KUKA KRL program: unicorn2_2.src

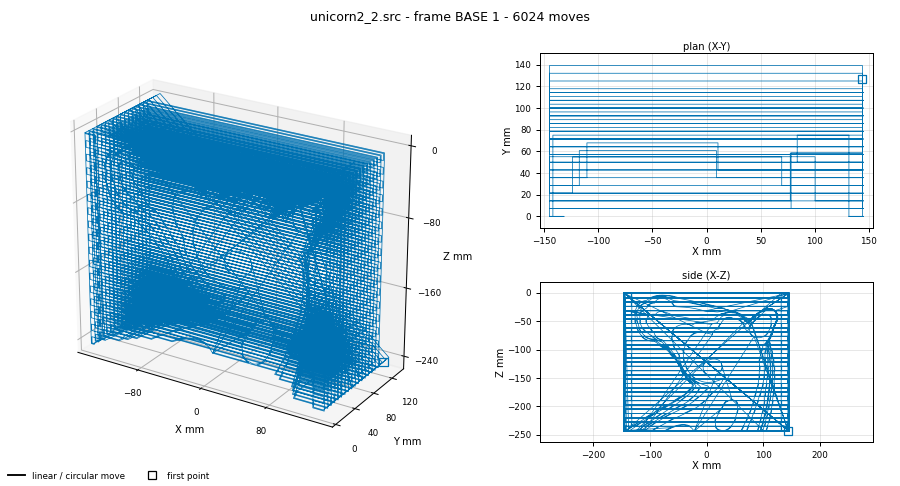
[picture p0: tool path of unicorn2_2.src in frame BASE 1, 6024 of 6025 moves have a stored position in this frame; points joined in program order, loops and branches not executed]
&ACCESS RVP
&REL 1
&PARAM TEMPLATE = C:\KRC\Roboter\Template\vorgabe
&PARAM EDITMASK = *
DEF unicorn2_2( )
EXT BAS (BAS_COMMAND :IN,REAL :IN )

INT INDX
FOR INDX=1 TO 6
	$ACC_AXIS[INDX]=50
	$VEL_AXIS[INDX]=20
ENDFOR

$VEL.ORI1=200
$VEL.ORI2=200
$ACC.ORI1=100
$ACC.ORI2=100

$VEL.CP = 0.2
$ACC.CP = 5

$IPO_MODE = #BASE
$APO.CDIS = 0.5
$ADVANCE = 5

$ACT_TOOL = 1
$TOOL=TOOL_DATA[1]
$ACT_BASE = 1
$BASE=BASE_DATA[1]

PTP {A1 -30.0,A2 -90.0,A3 90.0,A4 0.0,A5 90.0,A6 0.0}

LIN {X 144.015,Y 126.800,Z -242.561,A 90.000,B 90.000,C 0.000} C_DIS
LIN {X 144.015,Y 114.300,Z -242.561,A 90.000,B 90.000,C 0.000} C_DIS
LIN {X -144.015,Y 114.300,Z -242.561,A 90.000,B 90.000,C 0.000} C_DIS
LIN {X -144.015,Y 114.300,Z -235.012,A 90.000,B 90.000,C 0.000} C_DIS
LIN {X 144.015,Y 114.300,Z -235.012,A 90.000,B 90.000,C 0.000} C_DIS
LIN {X 144.015,Y 114.300,Z -227.464,A 90.000,B 90.000,C 0.000} C_DIS
LIN {X -144.015,Y 114.300,Z -227.464,A 90.000,B 90.000,C 0.000} C_DIS
LIN {X -144.015,Y 114.300,Z -219.915,A 90.000,B 90.000,C 0.000} C_DIS
LIN {X 144.015,Y 114.300,Z -219.915,A 90.000,B 90.000,C 0.000} C_DIS
LIN {X 144.015,Y 114.300,Z -212.366,A 90.000,B 90.000,C 0.000} C_DIS
LIN {X -144.015,Y 114.300,Z -212.366,A 90.000,B 90.000,C 0.000} C_DIS
LIN {X -144.015,Y 114.300,Z -204.817,A 90.000,B 90.000,C 0.000} C_DIS
LIN {X 144.015,Y 114.300,Z -204.817,A 90.000,B 90.000,C 0.000} C_DIS
LIN {X 144.015,Y 114.300,Z -197.269,A 90.000,B 90.000,C 0.000} C_DIS
LIN {X -144.015,Y 114.300,Z -197.269,A 90.000,B 90.000,C 0.000} C_DIS
LIN {X -144.015,Y 114.300,Z -189.720,A 90.000,B 90.000,C 0.000} C_DIS
LIN {X 144.015,Y 114.300,Z -189.720,A 90.000,B 90.000,C 0.000} C_DIS
LIN {X 144.015,Y 114.300,Z -182.171,A 90.000,B 90.000,C 0.000} C_DIS
LIN {X -144.015,Y 114.300,Z -182.171,A 90.000,B 90.000,C 0.000} C_DIS
LIN {X -144.015,Y 114.300,Z -174.622,A 90.000,B 90.000,C 0.000} C_DIS
LIN {X 144.015,Y 114.300,Z -174.622,A 90.000,B 90.000,C 0.000} C_DIS
LIN {X 144.015,Y 114.300,Z -167.073,A 90.000,B 90.000,C 0.000} C_DIS
LIN {X -144.015,Y 114.300,Z -167.073,A 90.000,B 90.000,C 0.000} C_DIS
LIN {X -144.015,Y 114.300,Z -159.525,A 90.000,B 90.000,C 0.000} C_DIS
LIN {X 144.015,Y 114.300,Z -159.525,A 90.000,B 90.000,C 0.000} C_DIS
LIN {X 144.015,Y 114.300,Z -151.976,A 90.000,B 90.000,C 0.000} C_DIS
LIN {X -144.015,Y 114.300,Z -151.976,A 90.000,B 90.000,C 0.000} C_DIS
LIN {X -144.015,Y 114.300,Z -144.427,A 90.000,B 90.000,C 0.000} C_DIS
LIN {X 144.015,Y 114.300,Z -144.427,A 90.000,B 90.000,C 0.000} C_DIS
LIN {X 144.015,Y 114.300,Z -136.878,A 90.000,B 90.000,C 0.000} C_DIS
LIN {X -144.015,Y 114.300,Z -136.878,A 90.000,B 90.000,C 0.000} C_DIS
LIN {X -144.015,Y 114.300,Z -129.329,A 90.000,B 90.000,C 0.000} C_DIS
LIN {X 144.015,Y 114.300,Z -129.329,A 90.000,B 90.000,C 0.000} C_DIS
LIN {X 144.015,Y 114.300,Z -121.781,A 90.000,B 90.000,C 0.000} C_DIS
LIN {X -144.015,Y 114.300,Z -121.781,A 90.000,B 90.000,C 0.000} C_DIS
LIN {X -144.015,Y 114.300,Z -114.232,A 90.000,B 90.000,C 0.000} C_DIS
LIN {X 144.015,Y 114.300,Z -114.232,A 90.000,B 90.000,C 0.000} C_DIS
LIN {X 144.015,Y 114.300,Z -106.683,A 90.000,B 90.000,C 0.000} C_DIS
LIN {X -144.015,Y 114.300,Z -106.683,A 90.000,B 90.000,C 0.000} C_DIS
LIN {X -144.015,Y 114.300,Z -99.134,A 90.000,B 90.000,C 0.000} C_DIS
LIN {X 144.015,Y 114.300,Z -99.134,A 90.000,B 90.000,C 0.000} C_DIS
LIN {X 144.015,Y 114.300,Z -91.586,A 90.000,B 90.000,C 0.000} C_DIS
LIN {X -144.015,Y 114.300,Z -91.586,A 90.000,B 90.000,C 0.000} C_DIS
LIN {X -144.015,Y 114.300,Z -84.037,A 90.000,B 90.000,C 0.000} C_DIS
LIN {X 144.015,Y 114.300,Z -84.037,A 90.000,B 90.000,C 0.000} C_DIS
LIN {X 144.015,Y 114.300,Z -76.488,A 90.000,B 90.000,C 0.000} C_DIS
LIN {X -144.015,Y 114.300,Z -76.488,A 90.000,B 90.000,C 0.000} C_DIS
LIN {X -144.015,Y 114.300,Z -68.939,A 90.000,B 90.000,C 0.000} C_DIS
LIN {X 144.015,Y 114.300,Z -68.939,A 90.000,B 90.000,C 0.000} C_DIS
LIN {X 144.015,Y 114.300,Z -61.390,A 90.000,B 90.000,C 0.000} C_DIS
LIN {X -144.015,Y 114.300,Z -61.390,A 90.000,B 90.000,C 0.000} C_DIS
LIN {X -144.015,Y 114.300,Z -53.842,A 90.000,B 90.000,C 0.000} C_DIS
LIN {X 144.015,Y 114.300,Z -53.842,A 90.000,B 90.000,C 0.000} C_DIS
LIN {X 144.015,Y 114.300,Z -46.293,A 90.000,B 90.000,C 0.000} C_DIS
LIN {X -144.015,Y 114.300,Z -46.293,A 90.000,B 90.000,C 0.000} C_DIS
LIN {X -144.015,Y 114.300,Z -38.744,A 90.000,B 90.000,C 0.000} C_DIS
LIN {X 144.015,Y 114.300,Z -38.744,A 90.000,B 90.000,C 0.000} C_DIS
LIN {X 144.015,Y 114.300,Z -31.195,A 90.000,B 90.000,C 0.000} C_DIS
LIN {X -144.015,Y 114.300,Z -31.195,A 90.000,B 90.000,C 0.000} C_DIS
LIN {X -144.015,Y 114.300,Z -23.646,A 90.000,B 90.000,C 0.000} C_DIS
LIN {X 144.015,Y 114.300,Z -23.646,A 90.000,B 90.000,C 0.000} C_DIS
LIN {X 144.015,Y 114.300,Z -16.098,A 90.000,B 90.000,C 0.000} C_DIS
LIN {X -144.015,Y 114.300,Z -16.098,A 90.000,B 90.000,C 0.000} C_DIS
LIN {X -144.015,Y 114.300,Z -8.549,A 90.000,B 90.000,C 0.000} C_DIS
LIN {X 144.015,Y 114.300,Z -8.549,A 90.000,B 90.000,C 0.000} C_DIS
LIN {X 144.015,Y 114.300,Z -1.000,A 90.000,B 90.000,C 0.000} C_DIS
LIN {X -144.015,Y 114.300,Z -1.000,A 90.000,B 90.000,C 0.000} C_DIS
LIN {X -145.015,Y 114.300,Z 0.000,A 90.000,B 90.000,C 0.000} C_DIS
LIN {X 145.015,Y 114.300,Z 0.000,A 90.000,B 90.000,C 0.000} C_DIS
LIN {X 145.015,Y 114.300,Z -243.561,A 90.000,B 90.000,C 0.000} C_DIS
LIN {X -145.015,Y 114.300,Z -243.561,A 90.000,B 90.000,C 0.000} C_DIS
LIN {X -145.015,Y 114.300,Z 0.000,A 90.000,B 90.000,C 0.000} C_DIS
LIN {X -145.015,Y 126.800,Z 0.000,A 90.000,B 90.000,C 0.000} C_DIS
LIN {X -145.015,Y 139.300,Z 0.000,A 90.000,B 90.000,C 0.000} C_DIS
LIN {X 144.015,Y 139.300,Z -242.561,A 90.000,B 90.000,C 0.000} C_DIS
LIN {X 144.015,Y 132.156,Z -242.561,A 90.000,B 90.000,C 0.000} C_DIS
LIN {X 144.015,Y 119.656,Z -242.561,A 90.000,B 90.000,C 0.000} C_DIS
LIN {X 144.015,Y 107.156,Z -242.561,A 90.000,B 90.000,C 0.000} C_DIS
LIN {X -144.015,Y 107.156,Z -242.561,A 90.000,B 90.000,C 0.000} C_DIS
LIN {X -144.015,Y 107.156,Z -235.012,A 90.000,B 90.000,C 0.000} C_DIS
LIN {X 144.015,Y 107.156,Z -235.012,A 90.000,B 90.000,C 0.000} C_DIS
LIN {X 144.015,Y 107.156,Z -227.464,A 90.000,B 90.000,C 0.000} C_DIS
LIN {X -144.015,Y 107.156,Z -227.464,A 90.000,B 90.000,C 0.000} C_DIS
LIN {X -144.015,Y 107.156,Z -219.915,A 90.000,B 90.000,C 0.000} C_DIS
LIN {X 144.015,Y 107.156,Z -219.915,A 90.000,B 90.000,C 0.000} C_DIS
LIN {X 144.015,Y 107.156,Z -212.366,A 90.000,B 90.000,C 0.000} C_DIS
LIN {X -144.015,Y 107.156,Z -212.366,A 90.000,B 90.000,C 0.000} C_DIS
LIN {X -144.015,Y 107.156,Z -204.817,A 90.000,B 90.000,C 0.000} C_DIS
LIN {X 144.015,Y 107.156,Z -204.817,A 90.000,B 90.000,C 0.000} C_DIS
LIN {X 144.015,Y 107.156,Z -197.269,A 90.000,B 90.000,C 0.000} C_DIS
LIN {X -144.015,Y 107.156,Z -197.269,A 90.000,B 90.000,C 0.000} C_DIS
LIN {X -144.015,Y 107.156,Z -189.720,A 90.000,B 90.000,C 0.000} C_DIS
LIN {X 144.015,Y 107.156,Z -189.720,A 90.000,B 90.000,C 0.000} C_DIS
LIN {X 144.015,Y 107.156,Z -182.171,A 90.000,B 90.000,C 0.000} C_DIS
LIN {X -144.015,Y 107.156,Z -182.171,A 90.000,B 90.000,C 0.000} C_DIS
LIN {X -144.015,Y 107.156,Z -174.622,A 90.000,B 90.000,C 0.000} C_DIS
LIN {X 144.015,Y 107.156,Z -174.622,A 90.000,B 90.000,C 0.000} C_DIS
LIN {X 144.015,Y 107.156,Z -167.073,A 90.000,B 90.000,C 0.000} C_DIS
LIN {X -144.015,Y 107.156,Z -167.073,A 90.000,B 90.000,C 0.000} C_DIS
LIN {X -144.015,Y 107.156,Z -159.525,A 90.000,B 90.000,C 0.000} C_DIS
LIN {X 144.015,Y 107.156,Z -159.525,A 90.000,B 90.000,C 0.000} C_DIS
LIN {X 144.015,Y 107.156,Z -151.976,A 90.000,B 90.000,C 0.000} C_DIS
LIN {X -144.015,Y 107.156,Z -151.976,A 90.000,B 90.000,C 0.000} C_DIS
LIN {X -144.015,Y 107.156,Z -144.427,A 90.000,B 90.000,C 0.000} C_DIS
LIN {X 144.015,Y 107.156,Z -144.427,A 90.000,B 90.000,C 0.000} C_DIS
LIN {X 144.015,Y 107.156,Z -136.878,A 90.000,B 90.000,C 0.000} C_DIS
LIN {X -144.015,Y 107.156,Z -136.878,A 90.000,B 90.000,C 0.000} C_DIS
LIN {X -144.015,Y 107.156,Z -129.329,A 90.000,B 90.000,C 0.000} C_DIS
LIN {X 144.015,Y 107.156,Z -129.329,A 90.000,B 90.000,C 0.000} C_DIS
LIN {X 144.015,Y 107.156,Z -121.781,A 90.000,B 90.000,C 0.000} C_DIS
LIN {X -144.015,Y 107.156,Z -121.781,A 90.000,B 90.000,C 0.000} C_DIS
LIN {X -144.015,Y 107.156,Z -114.232,A 90.000,B 90.000,C 0.000} C_DIS
LIN {X 144.015,Y 107.156,Z -114.232,A 90.000,B 90.000,C 0.000} C_DIS
LIN {X 144.015,Y 107.156,Z -106.683,A 90.000,B 90.000,C 0.000} C_DIS
LIN {X -144.015,Y 107.156,Z -106.683,A 90.000,B 90.000,C 0.000} C_DIS
LIN {X -144.015,Y 107.156,Z -99.134,A 90.000,B 90.000,C 0.000} C_DIS
LIN {X 144.015,Y 107.156,Z -99.134,A 90.000,B 90.000,C 0.000} C_DIS
LIN {X 144.015,Y 107.156,Z -91.586,A 90.000,B 90.000,C 0.000} C_DIS
LIN {X -144.015,Y 107.156,Z -91.586,A 90.000,B 90.000,C 0.000} C_DIS
LIN {X -144.015,Y 107.156,Z -84.037,A 90.000,B 90.000,C 0.000} C_DIS
LIN {X 144.015,Y 107.156,Z -84.037,A 90.000,B 90.000,C 0.000} C_DIS
LIN {X 144.015,Y 107.156,Z -76.488,A 90.000,B 90.000,C 0.000} C_DIS
LIN {X -144.015,Y 107.156,Z -76.488,A 90.000,B 90.000,C 0.000} C_DIS
LIN {X -144.015,Y 107.156,Z -68.939,A 90.000,B 90.000,C 0.000} C_DIS
LIN {X 144.015,Y 107.156,Z -68.939,A 90.000,B 90.000,C 0.000} C_DIS
LIN {X 144.015,Y 107.156,Z -61.390,A 90.000,B 90.000,C 0.000} C_DIS
LIN {X -144.015,Y 107.156,Z -61.390,A 90.000,B 90.000,C 0.000} C_DIS
LIN {X -144.015,Y 107.156,Z -53.842,A 90.000,B 90.000,C 0.000} C_DIS
LIN {X 144.015,Y 107.156,Z -53.842,A 90.000,B 90.000,C 0.000} C_DIS
LIN {X 144.015,Y 107.156,Z -46.293,A 90.000,B 90.000,C 0.000} C_DIS
LIN {X -144.015,Y 107.156,Z -46.293,A 90.000,B 90.000,C 0.000} C_DIS
LIN {X -144.015,Y 107.156,Z -38.744,A 90.000,B 90.000,C 0.000} C_DIS
LIN {X 144.015,Y 107.156,Z -38.744,A 90.000,B 90.000,C 0.000} C_DIS
LIN {X 144.015,Y 107.156,Z -31.195,A 90.000,B 90.000,C 0.000} C_DIS
LIN {X -144.015,Y 107.156,Z -31.195,A 90.000,B 90.000,C 0.000} C_DIS
LIN {X -144.015,Y 107.156,Z -23.646,A 90.000,B 90.000,C 0.000} C_DIS
LIN {X 144.015,Y 107.156,Z -23.646,A 90.000,B 90.000,C 0.000} C_DIS
LIN {X 144.015,Y 107.156,Z -16.098,A 90.000,B 90.000,C 0.000} C_DIS
LIN {X -144.015,Y 107.156,Z -16.098,A 90.000,B 90.000,C 0.000} C_DIS
LIN {X -144.015,Y 107.156,Z -8.549,A 90.000,B 90.000,C 0.000} C_DIS
LIN {X 144.015,Y 107.156,Z -8.549,A 90.000,B 90.000,C 0.000} C_DIS
LIN {X 144.015,Y 107.156,Z -1.000,A 90.000,B 90.000,C 0.000} C_DIS
LIN {X -144.015,Y 107.156,Z -1.000,A 90.000,B 90.000,C 0.000} C_DIS
LIN {X -145.015,Y 107.156,Z 0.000,A 90.000,B 90.000,C 0.000} C_DIS
LIN {X 145.015,Y 107.156,Z 0.000,A 90.000,B 90.000,C 0.000} C_DIS
LIN {X 145.015,Y 107.156,Z -243.561,A 90.000,B 90.000,C 0.000} C_DIS
LIN {X -145.015,Y 107.156,Z -243.561,A 90.000,B 90.000,C 0.000} C_DIS
LIN {X -145.015,Y 107.156,Z 0.000,A 90.000,B 90.000,C 0.000} C_DIS
LIN {X -145.015,Y 119.656,Z 0.000,A 90.000,B 90.000,C 0.000} C_DIS
LIN {X -145.015,Y 132.156,Z 0.000,A 90.000,B 90.000,C 0.000} C_DIS
LIN {X 144.015,Y 132.156,Z -242.561,A 90.000,B 90.000,C 0.000} C_DIS
LIN {X 144.015,Y 125.013,Z -242.561,A 90.000,B 90.000,C 0.000} C_DIS
LIN {X 144.015,Y 112.513,Z -242.561,A 90.000,B 90.000,C 0.000} C_DIS
LIN {X 144.015,Y 100.013,Z -242.561,A 90.000,B 90.000,C 0.000} C_DIS
LIN {X -144.015,Y 100.013,Z -242.561,A 90.000,B 90.000,C 0.000} C_DIS
LIN {X -144.015,Y 100.013,Z -235.012,A 90.000,B 90.000,C 0.000} C_DIS
LIN {X 144.015,Y 100.013,Z -235.012,A 90.000,B 90.000,C 0.000} C_DIS
LIN {X 144.015,Y 100.013,Z -227.464,A 90.000,B 90.000,C 0.000} C_DIS
LIN {X -144.015,Y 100.013,Z -227.464,A 90.000,B 90.000,C 0.000} C_DIS
LIN {X -144.015,Y 100.013,Z -219.915,A 90.000,B 90.000,C 0.000} C_DIS
LIN {X 144.015,Y 100.013,Z -219.915,A 90.000,B 90.000,C 0.000} C_DIS
LIN {X 144.015,Y 100.013,Z -212.366,A 90.000,B 90.000,C 0.000} C_DIS
LIN {X -144.015,Y 100.013,Z -212.366,A 90.000,B 90.000,C 0.000} C_DIS
LIN {X -144.015,Y 100.013,Z -204.817,A 90.000,B 90.000,C 0.000} C_DIS
LIN {X 144.015,Y 100.013,Z -204.817,A 90.000,B 90.000,C 0.000} C_DIS
LIN {X 144.015,Y 100.013,Z -197.269,A 90.000,B 90.000,C 0.000} C_DIS
LIN {X -144.015,Y 100.013,Z -197.269,A 90.000,B 90.000,C 0.000} C_DIS
LIN {X -144.015,Y 100.013,Z -189.720,A 90.000,B 90.000,C 0.000} C_DIS
LIN {X 144.015,Y 100.013,Z -189.720,A 90.000,B 90.000,C 0.000} C_DIS
LIN {X 144.015,Y 100.013,Z -182.171,A 90.000,B 90.000,C 0.000} C_DIS
LIN {X -144.015,Y 100.013,Z -182.171,A 90.000,B 90.000,C 0.000} C_DIS
LIN {X -144.015,Y 100.013,Z -174.622,A 90.000,B 90.000,C 0.000} C_DIS
LIN {X 144.015,Y 100.013,Z -174.622,A 90.000,B 90.000,C 0.000} C_DIS
LIN {X 144.015,Y 100.013,Z -167.073,A 90.000,B 90.000,C 0.000} C_DIS
LIN {X -144.015,Y 100.013,Z -167.073,A 90.000,B 90.000,C 0.000} C_DIS
LIN {X -144.015,Y 100.013,Z -159.525,A 90.000,B 90.000,C 0.000} C_DIS
LIN {X 144.015,Y 100.013,Z -159.525,A 90.000,B 90.000,C 0.000} C_DIS
LIN {X 144.015,Y 100.013,Z -151.976,A 90.000,B 90.000,C 0.000} C_DIS
LIN {X -144.015,Y 100.013,Z -151.976,A 90.000,B 90.000,C 0.000} C_DIS
LIN {X -144.015,Y 100.013,Z -144.427,A 90.000,B 90.000,C 0.000} C_DIS
LIN {X 144.015,Y 100.013,Z -144.427,A 90.000,B 90.000,C 0.000} C_DIS
LIN {X 144.015,Y 100.013,Z -136.878,A 90.000,B 90.000,C 0.000} C_DIS
LIN {X -144.015,Y 100.013,Z -136.878,A 90.000,B 90.000,C 0.000} C_DIS
LIN {X -144.015,Y 100.013,Z -129.329,A 90.000,B 90.000,C 0.000} C_DIS
LIN {X 144.015,Y 100.013,Z -129.329,A 90.000,B 90.000,C 0.000} C_DIS
LIN {X 144.015,Y 100.013,Z -121.781,A 90.000,B 90.000,C 0.000} C_DIS
LIN {X -144.015,Y 100.013,Z -121.781,A 90.000,B 90.000,C 0.000} C_DIS
LIN {X -144.015,Y 100.013,Z -114.232,A 90.000,B 90.000,C 0.000} C_DIS
LIN {X 144.015,Y 100.013,Z -114.232,A 90.000,B 90.000,C 0.000} C_DIS
LIN {X 144.015,Y 100.013,Z -106.683,A 90.000,B 90.000,C 0.000} C_DIS
LIN {X -144.015,Y 100.013,Z -106.683,A 90.000,B 90.000,C 0.000} C_DIS
LIN {X -144.015,Y 100.013,Z -99.134,A 90.000,B 90.000,C 0.000} C_DIS
LIN {X 144.015,Y 100.013,Z -99.134,A 90.000,B 90.000,C 0.000} C_DIS
LIN {X 144.015,Y 100.013,Z -91.586,A 90.000,B 90.000,C 0.000} C_DIS
LIN {X -144.015,Y 100.013,Z -91.586,A 90.000,B 90.000,C 0.000} C_DIS
LIN {X -144.015,Y 100.013,Z -84.037,A 90.000,B 90.000,C 0.000} C_DIS
LIN {X 144.015,Y 100.013,Z -84.037,A 90.000,B 90.000,C 0.000} C_DIS
LIN {X 144.015,Y 100.013,Z -76.488,A 90.000,B 90.000,C 0.000} C_DIS
LIN {X -144.015,Y 100.013,Z -76.488,A 90.000,B 90.000,C 0.000} C_DIS
LIN {X -144.015,Y 100.013,Z -68.939,A 90.000,B 90.000,C 0.000} C_DIS
LIN {X 144.015,Y 100.013,Z -68.939,A 90.000,B 90.000,C 0.000} C_DIS
LIN {X 144.015,Y 100.013,Z -61.390,A 90.000,B 90.000,C 0.000} C_DIS
LIN {X -144.015,Y 100.013,Z -61.390,A 90.000,B 90.000,C 0.000} C_DIS
LIN {X -144.015,Y 100.013,Z -53.842,A 90.000,B 90.000,C 0.000} C_DIS
LIN {X 144.015,Y 100.013,Z -53.842,A 90.000,B 90.000,C 0.000} C_DIS
LIN {X 144.015,Y 100.013,Z -46.293,A 90.000,B 90.000,C 0.000} C_DIS
LIN {X -144.015,Y 100.013,Z -46.293,A 90.000,B 90.000,C 0.000} C_DIS
LIN {X -144.015,Y 100.013,Z -38.744,A 90.000,B 90.000,C 0.000} C_DIS
LIN {X 144.015,Y 100.013,Z -38.744,A 90.000,B 90.000,C 0.000} C_DIS
LIN {X 144.015,Y 100.013,Z -31.195,A 90.000,B 90.000,C 0.000} C_DIS
LIN {X -144.015,Y 100.013,Z -31.195,A 90.000,B 90.000,C 0.000} C_DIS
LIN {X -144.015,Y 100.013,Z -23.646,A 90.000,B 90.000,C 0.000} C_DIS
LIN {X 144.015,Y 100.013,Z -23.646,A 90.000,B 90.000,C 0.000} C_DIS
LIN {X 144.015,Y 100.013,Z -16.098,A 90.000,B 90.000,C 0.000} C_DIS
LIN {X -144.015,Y 100.013,Z -16.098,A 90.000,B 90.000,C 0.000} C_DIS
LIN {X -144.015,Y 100.013,Z -8.549,A 90.000,B 90.000,C 0.000} C_DIS
LIN {X 144.015,Y 100.013,Z -8.549,A 90.000,B 90.000,C 0.000} C_DIS
LIN {X 144.015,Y 100.013,Z -1.000,A 90.000,B 90.000,C 0.000} C_DIS
LIN {X -144.015,Y 100.013,Z -1.000,A 90.000,B 90.000,C 0.000} C_DIS
LIN {X -145.015,Y 100.013,Z 0.000,A 90.000,B 90.000,C 0.000} C_DIS
LIN {X 145.015,Y 100.013,Z 0.000,A 90.000,B 90.000,C 0.000} C_DIS
LIN {X 145.015,Y 100.013,Z -243.561,A 90.000,B 90.000,C 0.000} C_DIS
LIN {X -145.015,Y 100.013,Z -243.561,A 90.000,B 90.000,C 0.000} C_DIS
LIN {X -145.015,Y 100.013,Z 0.000,A 90.000,B 90.000,C 0.000} C_DIS
LIN {X -145.015,Y 112.513,Z 0.000,A 90.000,B 90.000,C 0.000} C_DIS
LIN {X -145.015,Y 125.013,Z 0.000,A 90.000,B 90.000,C 0.000} C_DIS
LIN {X 144.015,Y 125.013,Z -242.561,A 90.000,B 90.000,C 0.000} C_DIS
LIN {X 144.015,Y 117.869,Z -242.561,A 90.000,B 90.000,C 0.000} C_DIS
LIN {X 144.015,Y 105.369,Z -242.561,A 90.000,B 90.000,C 0.000} C_DIS
LIN {X 144.015,Y 92.869,Z -242.561,A 90.000,B 90.000,C 0.000} C_DIS
LIN {X -144.015,Y 92.869,Z -242.561,A 90.000,B 90.000,C 0.000} C_DIS
LIN {X -144.015,Y 92.869,Z -235.012,A 90.000,B 90.000,C 0.000} C_DIS
LIN {X 144.015,Y 92.869,Z -235.012,A 90.000,B 90.000,C 0.000} C_DIS
LIN {X 144.015,Y 92.869,Z -227.464,A 90.000,B 90.000,C 0.000} C_DIS
LIN {X -144.015,Y 92.869,Z -227.464,A 90.000,B 90.000,C 0.000} C_DIS
LIN {X -144.015,Y 92.869,Z -219.915,A 90.000,B 90.000,C 0.000} C_DIS
LIN {X 144.015,Y 92.869,Z -219.915,A 90.000,B 90.000,C 0.000} C_DIS
LIN {X 144.015,Y 92.869,Z -212.366,A 90.000,B 90.000,C 0.000} C_DIS
LIN {X -144.015,Y 92.869,Z -212.366,A 90.000,B 90.000,C 0.000} C_DIS
LIN {X -144.015,Y 92.869,Z -204.817,A 90.000,B 90.000,C 0.000} C_DIS
LIN {X 144.015,Y 92.869,Z -204.817,A 90.000,B 90.000,C 0.000} C_DIS
LIN {X 144.015,Y 92.869,Z -197.269,A 90.000,B 90.000,C 0.000} C_DIS
LIN {X -144.015,Y 92.869,Z -197.269,A 90.000,B 90.000,C 0.000} C_DIS
LIN {X -144.015,Y 92.869,Z -189.720,A 90.000,B 90.000,C 0.000} C_DIS
LIN {X 144.015,Y 92.869,Z -189.720,A 90.000,B 90.000,C 0.000} C_DIS
LIN {X 144.015,Y 92.869,Z -182.171,A 90.000,B 90.000,C 0.000} C_DIS
LIN {X -144.015,Y 92.869,Z -182.171,A 90.000,B 90.000,C 0.000} C_DIS
LIN {X -144.015,Y 92.869,Z -174.622,A 90.000,B 90.000,C 0.000} C_DIS
LIN {X 144.015,Y 92.869,Z -174.622,A 90.000,B 90.000,C 0.000} C_DIS
LIN {X 144.015,Y 92.869,Z -167.073,A 90.000,B 90.000,C 0.000} C_DIS
LIN {X -144.015,Y 92.869,Z -167.073,A 90.000,B 90.000,C 0.000} C_DIS
LIN {X -144.015,Y 92.869,Z -159.525,A 90.000,B 90.000,C 0.000} C_DIS
LIN {X 144.015,Y 92.869,Z -159.525,A 90.000,B 90.000,C 0.000} C_DIS
LIN {X 144.015,Y 92.869,Z -151.976,A 90.000,B 90.000,C 0.000} C_DIS
LIN {X -144.015,Y 92.869,Z -151.976,A 90.000,B 90.000,C 0.000} C_DIS
LIN {X -144.015,Y 92.869,Z -144.427,A 90.000,B 90.000,C 0.000} C_DIS
LIN {X 144.015,Y 92.869,Z -144.427,A 90.000,B 90.000,C 0.000} C_DIS
LIN {X 144.015,Y 92.869,Z -136.878,A 90.000,B 90.000,C 0.000} C_DIS
LIN {X -144.015,Y 92.869,Z -136.878,A 90.000,B 90.000,C 0.000} C_DIS
LIN {X -144.015,Y 92.869,Z -129.329,A 90.000,B 90.000,C 0.000} C_DIS
LIN {X 144.015,Y 92.869,Z -129.329,A 90.000,B 90.000,C 0.000} C_DIS
LIN {X 144.015,Y 92.869,Z -121.781,A 90.000,B 90.000,C 0.000} C_DIS
LIN {X -144.015,Y 92.869,Z -121.781,A 90.000,B 90.000,C 0.000} C_DIS
LIN {X -144.015,Y 92.869,Z -114.232,A 90.000,B 90.000,C 0.000} C_DIS
LIN {X 144.015,Y 92.869,Z -114.232,A 90.000,B 90.000,C 0.000} C_DIS
LIN {X 144.015,Y 92.869,Z -106.683,A 90.000,B 90.000,C 0.000} C_DIS
LIN {X -144.015,Y 92.869,Z -106.683,A 90.000,B 90.000,C 0.000} C_DIS
LIN {X -144.015,Y 92.869,Z -99.134,A 90.000,B 90.000,C 0.000} C_DIS
LIN {X 144.015,Y 92.869,Z -99.134,A 90.000,B 90.000,C 0.000} C_DIS
LIN {X 144.015,Y 92.869,Z -91.586,A 90.000,B 90.000,C 0.000} C_DIS
LIN {X -144.015,Y 92.869,Z -91.586,A 90.000,B 90.000,C 0.000} C_DIS
LIN {X -144.015,Y 92.869,Z -84.037,A 90.000,B 90.000,C 0.000} C_DIS
LIN {X 144.015,Y 92.869,Z -84.037,A 90.000,B 90.000,C 0.000} C_DIS
LIN {X 144.015,Y 92.869,Z -76.488,A 90.000,B 90.000,C 0.000} C_DIS
LIN {X -144.015,Y 92.869,Z -76.488,A 90.000,B 90.000,C 0.000} C_DIS
LIN {X -144.015,Y 92.869,Z -68.939,A 90.000,B 90.000,C 0.000} C_DIS
LIN {X 144.015,Y 92.869,Z -68.939,A 90.000,B 90.000,C 0.000} C_DIS
LIN {X 144.015,Y 92.869,Z -61.390,A 90.000,B 90.000,C 0.000} C_DIS
LIN {X -144.015,Y 92.869,Z -61.390,A 90.000,B 90.000,C 0.000} C_DIS
LIN {X -144.015,Y 92.869,Z -53.842,A 90.000,B 90.000,C 0.000} C_DIS
LIN {X 144.015,Y 92.869,Z -53.842,A 90.000,B 90.000,C 0.000} C_DIS
LIN {X 144.015,Y 92.869,Z -46.293,A 90.000,B 90.000,C 0.000} C_DIS
LIN {X -144.015,Y 92.869,Z -46.293,A 90.000,B 90.000,C 0.000} C_DIS
LIN {X -144.015,Y 92.869,Z -38.744,A 90.000,B 90.000,C 0.000} C_DIS
LIN {X 144.015,Y 92.869,Z -38.744,A 90.000,B 90.000,C 0.000} C_DIS
LIN {X 144.015,Y 92.869,Z -31.195,A 90.000,B 90.000,C 0.000} C_DIS
LIN {X -144.015,Y 92.869,Z -31.195,A 90.000,B 90.000,C 0.000} C_DIS
LIN {X -144.015,Y 92.869,Z -23.646,A 90.000,B 90.000,C 0.000} C_DIS
LIN {X 144.015,Y 92.869,Z -23.646,A 90.000,B 90.000,C 0.000} C_DIS
LIN {X 144.015,Y 92.869,Z -16.098,A 90.000,B 90.000,C 0.000} C_DIS
LIN {X -144.015,Y 92.869,Z -16.098,A 90.000,B 90.000,C 0.000} C_DIS
LIN {X -144.015,Y 92.869,Z -8.549,A 90.000,B 90.000,C 0.000} C_DIS
LIN {X 144.015,Y 92.869,Z -8.549,A 90.000,B 90.000,C 0.000} C_DIS
LIN {X 144.015,Y 92.869,Z -1.000,A 90.000,B 90.000,C 0.000} C_DIS
LIN {X -144.015,Y 92.869,Z -1.000,A 90.000,B 90.000,C 0.000} C_DIS
LIN {X -145.015,Y 92.869,Z 0.000,A 90.000,B 90.000,C 0.000} C_DIS
LIN {X 145.015,Y 92.869,Z 0.000,A 90.000,B 90.000,C 0.000} C_DIS
LIN {X 145.015,Y 92.869,Z -243.561,A 90.000,B 90.000,C 0.000} C_DIS
LIN {X -145.015,Y 92.869,Z -243.561,A 90.000,B 90.000,C 0.000} C_DIS
LIN {X -145.015,Y 92.869,Z 0.000,A 90.000,B 90.000,C 0.000} C_DIS
LIN {X -145.015,Y 105.369,Z 0.000,A 90.000,B 90.000,C 0.000} C_DIS
LIN {X -145.015,Y 117.869,Z 0.000,A 90.000,B 90.000,C 0.000} C_DIS
LIN {X 144.015,Y 117.869,Z -242.561,A 90.000,B 90.000,C 0.000} C_DIS
LIN {X 144.015,Y 110.725,Z -242.561,A 90.000,B 90.000,C 0.000} C_DIS
LIN {X 144.015,Y 98.225,Z -242.561,A 90.000,B 90.000,C 0.000} C_DIS
LIN {X 144.015,Y 85.725,Z -242.561,A 90.000,B 90.000,C 0.000} C_DIS
LIN {X -144.015,Y 85.725,Z -242.561,A 90.000,B 90.000,C 0.000} C_DIS
LIN {X -144.015,Y 85.725,Z -235.012,A 90.000,B 90.000,C 0.000} C_DIS
LIN {X 144.015,Y 85.725,Z -235.012,A 90.000,B 90.000,C 0.000} C_DIS
LIN {X 144.015,Y 85.725,Z -227.464,A 90.000,B 90.000,C 0.000} C_DIS
LIN {X -144.015,Y 85.725,Z -227.464,A 90.000,B 90.000,C 0.000} C_DIS
LIN {X -144.015,Y 85.725,Z -219.915,A 90.000,B 90.000,C 0.000} C_DIS
LIN {X 144.015,Y 85.725,Z -219.915,A 90.000,B 90.000,C 0.000} C_DIS
LIN {X 144.015,Y 85.725,Z -212.366,A 90.000,B 90.000,C 0.000} C_DIS
LIN {X -144.015,Y 85.725,Z -212.366,A 90.000,B 90.000,C 0.000} C_DIS
LIN {X -144.015,Y 85.725,Z -204.817,A 90.000,B 90.000,C 0.000} C_DIS
LIN {X 144.015,Y 85.725,Z -204.817,A 90.000,B 90.000,C 0.000} C_DIS
LIN {X 144.015,Y 85.725,Z -197.269,A 90.000,B 90.000,C 0.000} C_DIS
LIN {X -144.015,Y 85.725,Z -197.269,A 90.000,B 90.000,C 0.000} C_DIS
LIN {X -144.015,Y 85.725,Z -189.720,A 90.000,B 90.000,C 0.000} C_DIS
LIN {X 144.015,Y 85.725,Z -189.720,A 90.000,B 90.000,C 0.000} C_DIS
LIN {X 144.015,Y 85.725,Z -182.171,A 90.000,B 90.000,C 0.000} C_DIS
LIN {X -144.015,Y 85.725,Z -182.171,A 90.000,B 90.000,C 0.000} C_DIS
LIN {X -144.015,Y 85.725,Z -174.622,A 90.000,B 90.000,C 0.000} C_DIS
LIN {X 144.015,Y 85.725,Z -174.622,A 90.000,B 90.000,C 0.000} C_DIS
LIN {X 144.015,Y 85.725,Z -167.073,A 90.000,B 90.000,C 0.000} C_DIS
LIN {X -144.015,Y 85.725,Z -167.073,A 90.000,B 90.000,C 0.000} C_DIS
LIN {X -144.015,Y 85.725,Z -159.525,A 90.000,B 90.000,C 0.000} C_DIS
LIN {X 144.015,Y 85.725,Z -159.525,A 90.000,B 90.000,C 0.000} C_DIS
LIN {X 144.015,Y 85.725,Z -151.976,A 90.000,B 90.000,C 0.000} C_DIS
LIN {X -144.015,Y 85.725,Z -151.976,A 90.000,B 90.000,C 0.000} C_DIS
LIN {X -144.015,Y 85.725,Z -144.427,A 90.000,B 90.000,C 0.000} C_DIS
LIN {X 144.015,Y 85.725,Z -144.427,A 90.000,B 90.000,C 0.000} C_DIS
LIN {X 144.015,Y 85.725,Z -136.878,A 90.000,B 90.000,C 0.000} C_DIS
LIN {X -144.015,Y 85.725,Z -136.878,A 90.000,B 90.000,C 0.000} C_DIS
LIN {X -144.015,Y 85.725,Z -129.329,A 90.000,B 90.000,C 0.000} C_DIS
LIN {X 144.015,Y 85.725,Z -129.329,A 90.000,B 90.000,C 0.000} C_DIS
LIN {X 144.015,Y 85.725,Z -121.781,A 90.000,B 90.000,C 0.000} C_DIS
LIN {X -144.015,Y 85.725,Z -121.781,A 90.000,B 90.000,C 0.000} C_DIS
LIN {X -144.015,Y 85.725,Z -114.232,A 90.000,B 90.000,C 0.000} C_DIS
LIN {X 144.015,Y 85.725,Z -114.232,A 90.000,B 90.000,C 0.000} C_DIS
LIN {X 144.015,Y 85.725,Z -106.683,A 90.000,B 90.000,C 0.000} C_DIS
LIN {X -144.015,Y 85.725,Z -106.683,A 90.000,B 90.000,C 0.000} C_DIS
LIN {X -144.015,Y 85.725,Z -99.134,A 90.000,B 90.000,C 0.000} C_DIS
LIN {X 144.015,Y 85.725,Z -99.134,A 90.000,B 90.000,C 0.000} C_DIS
LIN {X 144.015,Y 85.725,Z -91.586,A 90.000,B 90.000,C 0.000} C_DIS
LIN {X -144.015,Y 85.725,Z -91.586,A 90.000,B 90.000,C 0.000} C_DIS
LIN {X -144.015,Y 85.725,Z -84.037,A 90.000,B 90.000,C 0.000} C_DIS
LIN {X 144.015,Y 85.725,Z -84.037,A 90.000,B 90.000,C 0.000} C_DIS
LIN {X 144.015,Y 85.725,Z -76.488,A 90.000,B 90.000,C 0.000} C_DIS
LIN {X -144.015,Y 85.725,Z -76.488,A 90.000,B 90.000,C 0.000} C_DIS
LIN {X -144.015,Y 85.725,Z -68.939,A 90.000,B 90.000,C 0.000} C_DIS
LIN {X 144.015,Y 85.725,Z -68.939,A 90.000,B 90.000,C 0.000} C_DIS
LIN {X 144.015,Y 85.725,Z -61.390,A 90.000,B 90.000,C 0.000} C_DIS
LIN {X -144.015,Y 85.725,Z -61.390,A 90.000,B 90.000,C 0.000} C_DIS
LIN {X -144.015,Y 85.725,Z -53.842,A 90.000,B 90.000,C 0.000} C_DIS
LIN {X 144.015,Y 85.725,Z -53.842,A 90.000,B 90.000,C 0.000} C_DIS
LIN {X 144.015,Y 85.725,Z -46.293,A 90.000,B 90.000,C 0.000} C_DIS
LIN {X -144.015,Y 85.725,Z -46.293,A 90.000,B 90.000,C 0.000} C_DIS
LIN {X -144.015,Y 85.725,Z -38.744,A 90.000,B 90.000,C 0.000} C_DIS
LIN {X 144.015,Y 85.725,Z -38.744,A 90.000,B 90.000,C 0.000} C_DIS
LIN {X 144.015,Y 85.725,Z -31.195,A 90.000,B 90.000,C 0.000} C_DIS
LIN {X -144.015,Y 85.725,Z -31.195,A 90.000,B 90.000,C 0.000} C_DIS
LIN {X -144.015,Y 85.725,Z -23.646,A 90.000,B 90.000,C 0.000} C_DIS
LIN {X 144.015,Y 85.725,Z -23.646,A 90.000,B 90.000,C 0.000} C_DIS
LIN {X 144.015,Y 85.725,Z -16.098,A 90.000,B 90.000,C 0.000} C_DIS
LIN {X -144.015,Y 85.725,Z -16.098,A 90.000,B 90.000,C 0.000} C_DIS
LIN {X -144.015,Y 85.725,Z -8.549,A 90.000,B 90.000,C 0.000} C_DIS
LIN {X 144.015,Y 85.725,Z -8.549,A 90.000,B 90.000,C 0.000} C_DIS
LIN {X 144.015,Y 85.725,Z -1.000,A 90.000,B 90.000,C 0.000} C_DIS
LIN {X -144.015,Y 85.725,Z -1.000,A 90.000,B 90.000,C 0.000} C_DIS
LIN {X -145.015,Y 85.725,Z 0.000,A 90.000,B 90.000,C 0.000} C_DIS
LIN {X 145.015,Y 85.725,Z 0.000,A 90.000,B 90.000,C 0.000} C_DIS
LIN {X 145.015,Y 85.725,Z -243.561,A 90.000,B 90.000,C 0.000} C_DIS
LIN {X -145.015,Y 85.725,Z -243.561,A 90.000,B 90.000,C 0.000} C_DIS
LIN {X -145.015,Y 85.725,Z 0.000,A 90.000,B 90.000,C 0.000} C_DIS
LIN {X -145.015,Y 98.225,Z 0.000,A 90.000,B 90.000,C 0.000} C_DIS
LIN {X -145.015,Y 110.725,Z 0.000,A 90.000,B 90.000,C 0.000} C_DIS
LIN {X 144.015,Y 110.725,Z -242.561,A 90.000,B 90.000,C 0.000} C_DIS
LIN {X 144.015,Y 103.581,Z -242.561,A 90.000,B 90.000,C 0.000} C_DIS
LIN {X 144.015,Y 91.081,Z -242.561,A 90.000,B 90.000,C 0.000} C_DIS
LIN {X 144.015,Y 78.581,Z -242.561,A 90.000,B 90.000,C 0.000} C_DIS
LIN {X -144.015,Y 78.581,Z -242.561,A 90.000,B 90.000,C 0.000} C_DIS
LIN {X -144.015,Y 78.581,Z -235.012,A 90.000,B 90.000,C 0.000} C_DIS
LIN {X 144.015,Y 78.581,Z -235.012,A 90.000,B 90.000,C 0.000} C_DIS
LIN {X 144.015,Y 78.581,Z -227.464,A 90.000,B 90.000,C 0.000} C_DIS
LIN {X -144.015,Y 78.581,Z -227.464,A 90.000,B 90.000,C 0.000} C_DIS
LIN {X -144.015,Y 78.581,Z -219.915,A 90.000,B 90.000,C 0.000} C_DIS
LIN {X 144.015,Y 78.581,Z -219.915,A 90.000,B 90.000,C 0.000} C_DIS
LIN {X 144.015,Y 78.581,Z -212.366,A 90.000,B 90.000,C 0.000} C_DIS
LIN {X -144.015,Y 78.581,Z -212.366,A 90.000,B 90.000,C 0.000} C_DIS
LIN {X -144.015,Y 78.581,Z -204.817,A 90.000,B 90.000,C 0.000} C_DIS
LIN {X 144.015,Y 78.581,Z -204.817,A 90.000,B 90.000,C 0.000} C_DIS
LIN {X 144.015,Y 78.581,Z -197.269,A 90.000,B 90.000,C 0.000} C_DIS
LIN {X -144.015,Y 78.581,Z -197.269,A 90.000,B 90.000,C 0.000} C_DIS
LIN {X -144.015,Y 78.581,Z -189.720,A 90.000,B 90.000,C 0.000} C_DIS
LIN {X 144.015,Y 78.581,Z -189.720,A 90.000,B 90.000,C 0.000} C_DIS
LIN {X 144.015,Y 78.581,Z -182.171,A 90.000,B 90.000,C 0.000} C_DIS
LIN {X -144.015,Y 78.581,Z -182.171,A 90.000,B 90.000,C 0.000} C_DIS
LIN {X -144.015,Y 78.581,Z -174.622,A 90.000,B 90.000,C 0.000} C_DIS
LIN {X 144.015,Y 78.581,Z -174.622,A 90.000,B 90.000,C 0.000} C_DIS
LIN {X 144.015,Y 78.581,Z -167.073,A 90.000,B 90.000,C 0.000} C_DIS
LIN {X -144.015,Y 78.581,Z -167.073,A 90.000,B 90.000,C 0.000} C_DIS
LIN {X -144.015,Y 78.581,Z -159.525,A 90.000,B 90.000,C 0.000} C_DIS
LIN {X 144.015,Y 78.581,Z -159.525,A 90.000,B 90.000,C 0.000} C_DIS
LIN {X 144.015,Y 78.581,Z -151.976,A 90.000,B 90.000,C 0.000} C_DIS
LIN {X -144.015,Y 78.581,Z -151.976,A 90.000,B 90.000,C 0.000} C_DIS
LIN {X -144.015,Y 78.581,Z -144.427,A 90.000,B 90.000,C 0.000} C_DIS
LIN {X 144.015,Y 78.581,Z -144.427,A 90.000,B 90.000,C 0.000} C_DIS
LIN {X 144.015,Y 78.581,Z -136.878,A 90.000,B 90.000,C 0.000} C_DIS
LIN {X -144.015,Y 78.581,Z -136.878,A 90.000,B 90.000,C 0.000} C_DIS
LIN {X -144.015,Y 78.581,Z -129.329,A 90.000,B 90.000,C 0.000} C_DIS
LIN {X 144.015,Y 78.581,Z -129.329,A 90.000,B 90.000,C 0.000} C_DIS
LIN {X 144.015,Y 78.581,Z -121.781,A 90.000,B 90.000,C 0.000} C_DIS
LIN {X -144.015,Y 78.581,Z -121.781,A 90.000,B 90.000,C 0.000} C_DIS
LIN {X -144.015,Y 78.581,Z -114.232,A 90.000,B 90.000,C 0.000} C_DIS
LIN {X 144.015,Y 78.581,Z -114.232,A 90.000,B 90.000,C 0.000} C_DIS
LIN {X 144.015,Y 78.581,Z -106.683,A 90.000,B 90.000,C 0.000} C_DIS
LIN {X -144.015,Y 78.581,Z -106.683,A 90.000,B 90.000,C 0.000} C_DIS
LIN {X -144.015,Y 78.581,Z -99.134,A 90.000,B 90.000,C 0.000} C_DIS
LIN {X 144.015,Y 78.581,Z -99.134,A 90.000,B 90.000,C 0.000} C_DIS
LIN {X 144.015,Y 78.581,Z -91.586,A 90.000,B 90.000,C 0.000} C_DIS
LIN {X -144.015,Y 78.581,Z -91.586,A 90.000,B 90.000,C 0.000} C_DIS
LIN {X -144.015,Y 78.581,Z -84.037,A 90.000,B 90.000,C 0.000} C_DIS
LIN {X 144.015,Y 78.581,Z -84.037,A 90.000,B 90.000,C 0.000} C_DIS
LIN {X 144.015,Y 78.581,Z -76.488,A 90.000,B 90.000,C 0.000} C_DIS
LIN {X -144.015,Y 78.581,Z -76.488,A 90.000,B 90.000,C 0.000} C_DIS
LIN {X -144.015,Y 78.581,Z -68.939,A 90.000,B 90.000,C 0.000} C_DIS
LIN {X 144.015,Y 78.581,Z -68.939,A 90.000,B 90.000,C 0.000} C_DIS
LIN {X 144.015,Y 78.581,Z -61.390,A 90.000,B 90.000,C 0.000} C_DIS
LIN {X -144.015,Y 78.581,Z -61.390,A 90.000,B 90.000,C 0.000} C_DIS
LIN {X -144.015,Y 78.581,Z -53.842,A 90.000,B 90.000,C 0.000} C_DIS
LIN {X 144.015,Y 78.581,Z -53.842,A 90.000,B 90.000,C 0.000} C_DIS
LIN {X 144.015,Y 78.581,Z -46.293,A 90.000,B 90.000,C 0.000} C_DIS
LIN {X -144.015,Y 78.581,Z -46.293,A 90.000,B 90.000,C 0.000} C_DIS
LIN {X -144.015,Y 78.581,Z -38.744,A 90.000,B 90.000,C 0.000} C_DIS
LIN {X 144.015,Y 78.581,Z -38.744,A 90.000,B 90.000,C 0.000} C_DIS
LIN {X 144.015,Y 78.581,Z -31.195,A 90.000,B 90.000,C 0.000} C_DIS
LIN {X -144.015,Y 78.581,Z -31.195,A 90.000,B 90.000,C 0.000} C_DIS
LIN {X -144.015,Y 78.581,Z -23.646,A 90.000,B 90.000,C 0.000} C_DIS
LIN {X 144.015,Y 78.581,Z -23.646,A 90.000,B 90.000,C 0.000} C_DIS
LIN {X 144.015,Y 78.581,Z -16.098,A 90.000,B 90.000,C 0.000} C_DIS
LIN {X -144.015,Y 78.581,Z -16.098,A 90.000,B 90.000,C 0.000} C_DIS
LIN {X -144.015,Y 78.581,Z -8.549,A 90.000,B 90.000,C 0.000} C_DIS
LIN {X 144.015,Y 78.581,Z -8.549,A 90.000,B 90.000,C 0.000} C_DIS
LIN {X 144.015,Y 78.581,Z -1.000,A 90.000,B 90.000,C 0.000} C_DIS
LIN {X -144.015,Y 78.581,Z -1.000,A 90.000,B 90.000,C 0.000} C_DIS
LIN {X -145.015,Y 78.581,Z 0.000,A 90.000,B 90.000,C 0.000} C_DIS
LIN {X 145.015,Y 78.581,Z 0.000,A 90.000,B 90.000,C 0.000} C_DIS
LIN {X 145.015,Y 78.581,Z -243.561,A 90.000,B 90.000,C 0.000} C_DIS
LIN {X -145.015,Y 78.581,Z -243.561,A 90.000,B 90.000,C 0.000} C_DIS
LIN {X -145.015,Y 78.581,Z 0.000,A 90.000,B 90.000,C 0.000} C_DIS
LIN {X -145.015,Y 91.081,Z 0.000,A 90.000,B 90.000,C 0.000} C_DIS
LIN {X -145.015,Y 103.581,Z 0.000,A 90.000,B 90.000,C 0.000} C_DIS
LIN {X 144.015,Y 103.581,Z -242.561,A 90.000,B 90.000,C 0.000} C_DIS
LIN {X 144.015,Y 96.438,Z -242.561,A 90.000,B 90.000,C 0.000} C_DIS
LIN {X 144.015,Y 83.938,Z -242.561,A 90.000,B 90.000,C 0.000} C_DIS
LIN {X 144.015,Y 71.438,Z -242.561,A 90.000,B 90.000,C 0.000} C_DIS
LIN {X -144.015,Y 71.438,Z -242.561,A 90.000,B 90.000,C 0.000} C_DIS
LIN {X -144.015,Y 71.438,Z -235.012,A 90.000,B 90.000,C 0.000} C_DIS
LIN {X 144.015,Y 71.438,Z -235.012,A 90.000,B 90.000,C 0.000} C_DIS
LIN {X 144.015,Y 71.438,Z -227.464,A 90.000,B 90.000,C 0.000} C_DIS
LIN {X -144.015,Y 71.438,Z -227.464,A 90.000,B 90.000,C 0.000} C_DIS
LIN {X -144.015,Y 71.438,Z -219.915,A 90.000,B 90.000,C 0.000} C_DIS
LIN {X 144.015,Y 71.438,Z -219.915,A 90.000,B 90.000,C 0.000} C_DIS
LIN {X 144.015,Y 71.438,Z -212.366,A 90.000,B 90.000,C 0.000} C_DIS
LIN {X -144.015,Y 71.438,Z -212.366,A 90.000,B 90.000,C 0.000} C_DIS
LIN {X -144.015,Y 71.438,Z -204.817,A 90.000,B 90.000,C 0.000} C_DIS
LIN {X 144.015,Y 71.438,Z -204.817,A 90.000,B 90.000,C 0.000} C_DIS
LIN {X 144.015,Y 71.438,Z -197.269,A 90.000,B 90.000,C 0.000} C_DIS
LIN {X -144.015,Y 71.438,Z -197.269,A 90.000,B 90.000,C 0.000} C_DIS
LIN {X -144.015,Y 71.438,Z -189.720,A 90.000,B 90.000,C 0.000} C_DIS
LIN {X 144.015,Y 71.438,Z -189.720,A 90.000,B 90.000,C 0.000} C_DIS
LIN {X 144.015,Y 71.438,Z -182.171,A 90.000,B 90.000,C 0.000} C_DIS
LIN {X -144.015,Y 71.438,Z -182.171,A 90.000,B 90.000,C 0.000} C_DIS
LIN {X -144.015,Y 71.438,Z -174.622,A 90.000,B 90.000,C 0.000} C_DIS
LIN {X 144.015,Y 71.438,Z -174.622,A 90.000,B 90.000,C 0.000} C_DIS
LIN {X 144.015,Y 71.438,Z -167.073,A 90.000,B 90.000,C 0.000} C_DIS
LIN {X -144.015,Y 71.438,Z -167.073,A 90.000,B 90.000,C 0.000} C_DIS
LIN {X -144.015,Y 71.438,Z -159.525,A 90.000,B 90.000,C 0.000} C_DIS
LIN {X 144.015,Y 71.438,Z -159.525,A 90.000,B 90.000,C 0.000} C_DIS
LIN {X 144.015,Y 71.438,Z -151.976,A 90.000,B 90.000,C 0.000} C_DIS
LIN {X -144.015,Y 71.438,Z -151.976,A 90.000,B 90.000,C 0.000} C_DIS
LIN {X -144.015,Y 71.438,Z -144.427,A 90.000,B 90.000,C 0.000} C_DIS
LIN {X 144.015,Y 71.438,Z -144.427,A 90.000,B 90.000,C 0.000} C_DIS
LIN {X 144.015,Y 71.438,Z -136.878,A 90.000,B 90.000,C 0.000} C_DIS
LIN {X -144.015,Y 71.438,Z -136.878,A 90.000,B 90.000,C 0.000} C_DIS
LIN {X -144.015,Y 71.438,Z -129.329,A 90.000,B 90.000,C 0.000} C_DIS
LIN {X 144.015,Y 71.438,Z -129.329,A 90.000,B 90.000,C 0.000} C_DIS
LIN {X 144.015,Y 71.438,Z -121.781,A 90.000,B 90.000,C 0.000} C_DIS
LIN {X -144.015,Y 71.438,Z -121.781,A 90.000,B 90.000,C 0.000} C_DIS
LIN {X -144.015,Y 71.438,Z -114.232,A 90.000,B 90.000,C 0.000} C_DIS
LIN {X 144.015,Y 71.438,Z -114.232,A 90.000,B 90.000,C 0.000} C_DIS
LIN {X 144.015,Y 71.438,Z -106.683,A 90.000,B 90.000,C 0.000} C_DIS
LIN {X -144.015,Y 71.438,Z -106.683,A 90.000,B 90.000,C 0.000} C_DIS
LIN {X -144.015,Y 71.438,Z -99.134,A 90.000,B 90.000,C 0.000} C_DIS
LIN {X 144.015,Y 71.438,Z -99.134,A 90.000,B 90.000,C 0.000} C_DIS
LIN {X 144.015,Y 71.438,Z -91.586,A 90.000,B 90.000,C 0.000} C_DIS
LIN {X -144.015,Y 71.438,Z -91.586,A 90.000,B 90.000,C 0.000} C_DIS
LIN {X -144.015,Y 71.438,Z -84.037,A 90.000,B 90.000,C 0.000} C_DIS
LIN {X 144.015,Y 71.438,Z -84.037,A 90.000,B 90.000,C 0.000} C_DIS
LIN {X 144.015,Y 71.438,Z -76.488,A 90.000,B 90.000,C 0.000} C_DIS
LIN {X -144.015,Y 71.438,Z -76.488,A 90.000,B 90.000,C 0.000} C_DIS
LIN {X -144.015,Y 71.438,Z -68.939,A 90.000,B 90.000,C 0.000} C_DIS
LIN {X 144.015,Y 71.438,Z -68.939,A 90.000,B 90.000,C 0.000} C_DIS
LIN {X 144.015,Y 71.438,Z -61.390,A 90.000,B 90.000,C 0.000} C_DIS
LIN {X -144.015,Y 71.438,Z -61.390,A 90.000,B 90.000,C 0.000} C_DIS
LIN {X -144.015,Y 71.438,Z -53.842,A 90.000,B 90.000,C 0.000} C_DIS
LIN {X 144.015,Y 71.438,Z -53.842,A 90.000,B 90.000,C 0.000} C_DIS
LIN {X 144.015,Y 71.438,Z -46.293,A 90.000,B 90.000,C 0.000} C_DIS
LIN {X -144.015,Y 71.438,Z -46.293,A 90.000,B 90.000,C 0.000} C_DIS
LIN {X -144.015,Y 71.438,Z -38.744,A 90.000,B 90.000,C 0.000} C_DIS
LIN {X 144.015,Y 71.438,Z -38.744,A 90.000,B 90.000,C 0.000} C_DIS
LIN {X 144.015,Y 71.438,Z -31.195,A 90.000,B 90.000,C 0.000} C_DIS
LIN {X -144.015,Y 71.438,Z -31.195,A 90.000,B 90.000,C 0.000} C_DIS
LIN {X -144.015,Y 71.438,Z -23.646,A 90.000,B 90.000,C 0.000} C_DIS
LIN {X 144.015,Y 71.438,Z -23.646,A 90.000,B 90.000,C 0.000} C_DIS
LIN {X 144.015,Y 71.438,Z -16.098,A 90.000,B 90.000,C 0.000} C_DIS
LIN {X -144.015,Y 71.438,Z -16.098,A 90.000,B 90.000,C 0.000} C_DIS
LIN {X -144.015,Y 71.438,Z -8.549,A 90.000,B 90.000,C 0.000} C_DIS
LIN {X 144.015,Y 71.438,Z -8.549,A 90.000,B 90.000,C 0.000} C_DIS
LIN {X 144.015,Y 71.438,Z -1.000,A 90.000,B 90.000,C 0.000} C_DIS
LIN {X -144.015,Y 71.438,Z -1.000,A 90.000,B 90.000,C 0.000} C_DIS
LIN {X -145.015,Y 71.438,Z 0.000,A 90.000,B 90.000,C 0.000} C_DIS
LIN {X 145.015,Y 71.438,Z 0.000,A 90.000,B 90.000,C 0.000} C_DIS
LIN {X 145.015,Y 71.438,Z -243.561,A 90.000,B 90.000,C 0.000} C_DIS
LIN {X -145.015,Y 71.438,Z -243.561,A 90.000,B 90.000,C 0.000} C_DIS
LIN {X -145.015,Y 71.438,Z 0.000,A 90.000,B 90.000,C 0.000} C_DIS
LIN {X -145.015,Y 83.938,Z 0.000,A 90.000,B 90.000,C 0.000} C_DIS
LIN {X -145.015,Y 96.438,Z 0.000,A 90.000,B 90.000,C 0.000} C_DIS
LIN {X 144.015,Y 96.438,Z -242.561,A 90.000,B 90.000,C 0.000} C_DIS
LIN {X 144.015,Y 89.294,Z -242.561,A 90.000,B 90.000,C 0.000} C_DIS
LIN {X 144.015,Y 76.794,Z -242.561,A 90.000,B 90.000,C 0.000} C_DIS
LIN {X 144.015,Y 64.294,Z -242.561,A 90.000,B 90.000,C 0.000} C_DIS
LIN {X -144.015,Y 64.294,Z -242.561,A 90.000,B 90.000,C 0.000} C_DIS
LIN {X -144.015,Y 64.294,Z -235.012,A 90.000,B 90.000,C 0.000} C_DIS
LIN {X 144.015,Y 64.294,Z -235.012,A 90.000,B 90.000,C 0.000} C_DIS
LIN {X 144.015,Y 64.294,Z -227.464,A 90.000,B 90.000,C 0.000} C_DIS
LIN {X -144.015,Y 64.294,Z -227.464,A 90.000,B 90.000,C 0.000} C_DIS
LIN {X -144.015,Y 64.294,Z -219.915,A 90.000,B 90.000,C 0.000} C_DIS
LIN {X 144.015,Y 64.294,Z -219.915,A 90.000,B 90.000,C 0.000} C_DIS
LIN {X 144.015,Y 64.294,Z -212.366,A 90.000,B 90.000,C 0.000} C_DIS
LIN {X -144.015,Y 64.294,Z -212.366,A 90.000,B 90.000,C 0.000} C_DIS
LIN {X -144.015,Y 64.294,Z -204.817,A 90.000,B 90.000,C 0.000} C_DIS
LIN {X 144.015,Y 64.294,Z -204.817,A 90.000,B 90.000,C 0.000} C_DIS
LIN {X 144.015,Y 64.294,Z -197.269,A 90.000,B 90.000,C 0.000} C_DIS
LIN {X -144.015,Y 64.294,Z -197.269,A 90.000,B 90.000,C 0.000} C_DIS
LIN {X -144.015,Y 64.294,Z -189.720,A 90.000,B 90.000,C 0.000} C_DIS
LIN {X 144.015,Y 64.294,Z -189.720,A 90.000,B 90.000,C 0.000} C_DIS
LIN {X 144.015,Y 64.294,Z -182.171,A 90.000,B 90.000,C 0.000} C_DIS
LIN {X -144.015,Y 64.294,Z -182.171,A 90.000,B 90.000,C 0.000} C_DIS
LIN {X -144.015,Y 64.294,Z -174.622,A 90.000,B 90.000,C 0.000} C_DIS
LIN {X 144.015,Y 64.294,Z -174.622,A 90.000,B 90.000,C 0.000} C_DIS
LIN {X 144.015,Y 64.294,Z -167.073,A 90.000,B 90.000,C 0.000} C_DIS
LIN {X -144.015,Y 64.294,Z -167.073,A 90.000,B 90.000,C 0.000} C_DIS
LIN {X -144.015,Y 64.294,Z -159.525,A 90.000,B 90.000,C 0.000} C_DIS
LIN {X 144.015,Y 64.294,Z -159.525,A 90.000,B 90.000,C 0.000} C_DIS
LIN {X 144.015,Y 64.294,Z -151.976,A 90.000,B 90.000,C 0.000} C_DIS
LIN {X -144.015,Y 64.294,Z -151.976,A 90.000,B 90.000,C 0.000} C_DIS
LIN {X -144.015,Y 64.294,Z -144.427,A 90.000,B 90.000,C 0.000} C_DIS
LIN {X 144.015,Y 64.294,Z -144.427,A 90.000,B 90.000,C 0.000} C_DIS
LIN {X 144.015,Y 64.294,Z -136.878,A 90.000,B 90.000,C 0.000} C_DIS
LIN {X -144.015,Y 64.294,Z -136.878,A 90.000,B 90.000,C 0.000} C_DIS
LIN {X -144.015,Y 64.294,Z -129.329,A 90.000,B 90.000,C 0.000} C_DIS
LIN {X 144.015,Y 64.294,Z -129.329,A 90.000,B 90.000,C 0.000} C_DIS
LIN {X 144.015,Y 64.294,Z -121.781,A 90.000,B 90.000,C 0.000} C_DIS
LIN {X -144.015,Y 64.294,Z -121.781,A 90.000,B 90.000,C 0.000} C_DIS
LIN {X -144.015,Y 64.294,Z -114.232,A 90.000,B 90.000,C 0.000} C_DIS
LIN {X 144.015,Y 64.294,Z -114.232,A 90.000,B 90.000,C 0.000} C_DIS
LIN {X 144.015,Y 64.294,Z -106.683,A 90.000,B 90.000,C 0.000} C_DIS
LIN {X -144.015,Y 64.294,Z -106.683,A 90.000,B 90.000,C 0.000} C_DIS
LIN {X -144.015,Y 64.294,Z -99.134,A 90.000,B 90.000,C 0.000} C_DIS
LIN {X 144.015,Y 64.294,Z -99.134,A 90.000,B 90.000,C 0.000} C_DIS
LIN {X 144.015,Y 64.294,Z -91.586,A 90.000,B 90.000,C 0.000} C_DIS
LIN {X -144.015,Y 64.294,Z -91.586,A 90.000,B 90.000,C 0.000} C_DIS
LIN {X -144.015,Y 64.294,Z -84.037,A 90.000,B 90.000,C 0.000} C_DIS
LIN {X 144.015,Y 64.294,Z -84.037,A 90.000,B 90.000,C 0.000} C_DIS
LIN {X 144.015,Y 64.294,Z -76.488,A 90.000,B 90.000,C 0.000} C_DIS
LIN {X -144.015,Y 64.294,Z -76.488,A 90.000,B 90.000,C 0.000} C_DIS
LIN {X -144.015,Y 64.294,Z -68.939,A 90.000,B 90.000,C 0.000} C_DIS
LIN {X 144.015,Y 64.294,Z -68.939,A 90.000,B 90.000,C 0.000} C_DIS
LIN {X 144.015,Y 64.294,Z -61.390,A 90.000,B 90.000,C 0.000} C_DIS
LIN {X -144.015,Y 64.294,Z -61.390,A 90.000,B 90.000,C 0.000} C_DIS
LIN {X -144.015,Y 64.294,Z -53.842,A 90.000,B 90.000,C 0.000} C_DIS
LIN {X 144.015,Y 64.294,Z -53.842,A 90.000,B 90.000,C 0.000} C_DIS
LIN {X 144.015,Y 64.294,Z -46.293,A 90.000,B 90.000,C 0.000} C_DIS
LIN {X -144.015,Y 64.294,Z -46.293,A 90.000,B 90.000,C 0.000} C_DIS
LIN {X -144.015,Y 64.294,Z -38.744,A 90.000,B 90.000,C 0.000} C_DIS
LIN {X 144.015,Y 64.294,Z -38.744,A 90.000,B 90.000,C 0.000} C_DIS
LIN {X 144.015,Y 64.294,Z -31.195,A 90.000,B 90.000,C 0.000} C_DIS
LIN {X -144.015,Y 64.294,Z -31.195,A 90.000,B 90.000,C 0.000} C_DIS
LIN {X -144.015,Y 64.294,Z -23.646,A 90.000,B 90.000,C 0.000} C_DIS
LIN {X 144.015,Y 64.294,Z -23.646,A 90.000,B 90.000,C 0.000} C_DIS
LIN {X 144.015,Y 64.294,Z -16.098,A 90.000,B 90.000,C 0.000} C_DIS
LIN {X -144.015,Y 64.294,Z -16.098,A 90.000,B 90.000,C 0.000} C_DIS
LIN {X -144.015,Y 64.294,Z -8.549,A 90.000,B 90.000,C 0.000} C_DIS
LIN {X 144.015,Y 64.294,Z -8.549,A 90.000,B 90.000,C 0.000} C_DIS
LIN {X 144.015,Y 64.294,Z -1.000,A 90.000,B 90.000,C 0.000} C_DIS
LIN {X -144.015,Y 64.294,Z -1.000,A 90.000,B 90.000,C 0.000} C_DIS
LIN {X -145.015,Y 64.294,Z 0.000,A 90.000,B 90.000,C 0.000} C_DIS
LIN {X 145.015,Y 64.294,Z 0.000,A 90.000,B 90.000,C 0.000} C_DIS
LIN {X 145.015,Y 64.294,Z -243.561,A 90.000,B 90.000,C 0.000} C_DIS
LIN {X -145.015,Y 64.294,Z -243.561,A 90.000,B 90.000,C 0.000} C_DIS
LIN {X -145.015,Y 64.294,Z 0.000,A 90.000,B 90.000,C 0.000} C_DIS
LIN {X -145.015,Y 76.794,Z 0.000,A 90.000,B 90.000,C 0.000} C_DIS
LIN {X -145.015,Y 89.294,Z 0.000,A 90.000,B 90.000,C 0.000} C_DIS
LIN {X 144.015,Y 89.294,Z -242.561,A 90.000,B 90.000,C 0.000} C_DIS
LIN {X 144.015,Y 82.150,Z -242.561,A 90.000,B 90.000,C 0.000} C_DIS
LIN {X 144.015,Y 69.650,Z -242.561,A 90.000,B 90.000,C 0.000} C_DIS
LIN {X 144.015,Y 57.150,Z -242.561,A 90.000,B 90.000,C 0.000} C_DIS
LIN {X -144.015,Y 57.150,Z -242.561,A 90.000,B 90.000,C 0.000} C_DIS
LIN {X -144.015,Y 57.150,Z -235.012,A 90.000,B 90.000,C 0.000} C_DIS
LIN {X 144.015,Y 57.150,Z -235.012,A 90.000,B 90.000,C 0.000} C_DIS
LIN {X 144.015,Y 57.150,Z -227.464,A 90.000,B 90.000,C 0.000} C_DIS
LIN {X -144.015,Y 57.150,Z -227.464,A 90.000,B 90.000,C 0.000} C_DIS
LIN {X -144.015,Y 57.150,Z -219.915,A 90.000,B 90.000,C 0.000} C_DIS
LIN {X 144.015,Y 57.150,Z -219.915,A 90.000,B 90.000,C 0.000} C_DIS
LIN {X 144.015,Y 57.150,Z -212.366,A 90.000,B 90.000,C 0.000} C_DIS
LIN {X -144.015,Y 57.150,Z -212.366,A 90.000,B 90.000,C 0.000} C_DIS
LIN {X -144.015,Y 57.150,Z -204.817,A 90.000,B 90.000,C 0.000} C_DIS
LIN {X 144.015,Y 57.150,Z -204.817,A 90.000,B 90.000,C 0.000} C_DIS
LIN {X 144.015,Y 57.150,Z -197.269,A 90.000,B 90.000,C 0.000} C_DIS
LIN {X -144.015,Y 57.150,Z -197.269,A 90.000,B 90.000,C 0.000} C_DIS
LIN {X -144.015,Y 57.150,Z -189.720,A 90.000,B 90.000,C 0.000} C_DIS
LIN {X 144.015,Y 57.150,Z -189.720,A 90.000,B 90.000,C 0.000} C_DIS
LIN {X 144.015,Y 57.150,Z -182.171,A 90.000,B 90.000,C 0.000} C_DIS
LIN {X -144.015,Y 57.150,Z -182.171,A 90.000,B 90.000,C 0.000} C_DIS
LIN {X -144.015,Y 57.150,Z -174.622,A 90.000,B 90.000,C 0.000} C_DIS
LIN {X 144.015,Y 57.150,Z -174.622,A 90.000,B 90.000,C 0.000} C_DIS
LIN {X 144.015,Y 57.150,Z -167.073,A 90.000,B 90.000,C 0.000} C_DIS
LIN {X -144.015,Y 57.150,Z -167.073,A 90.000,B 90.000,C 0.000} C_DIS
LIN {X -144.015,Y 57.150,Z -159.525,A 90.000,B 90.000,C 0.000} C_DIS
LIN {X 144.015,Y 57.150,Z -159.525,A 90.000,B 90.000,C 0.000} C_DIS
LIN {X 144.015,Y 57.150,Z -151.976,A 90.000,B 90.000,C 0.000} C_DIS
LIN {X -144.015,Y 57.150,Z -151.976,A 90.000,B 90.000,C 0.000} C_DIS
LIN {X -144.015,Y 57.150,Z -144.427,A 90.000,B 90.000,C 0.000} C_DIS
LIN {X 144.015,Y 57.150,Z -144.427,A 90.000,B 90.000,C 0.000} C_DIS
LIN {X 144.015,Y 57.150,Z -136.878,A 90.000,B 90.000,C 0.000} C_DIS
LIN {X -144.015,Y 57.150,Z -136.878,A 90.000,B 90.000,C 0.000} C_DIS
LIN {X -144.015,Y 57.150,Z -129.329,A 90.000,B 90.000,C 0.000} C_DIS
LIN {X 144.015,Y 57.150,Z -129.329,A 90.000,B 90.000,C 0.000} C_DIS
LIN {X 144.015,Y 57.150,Z -121.781,A 90.000,B 90.000,C 0.000} C_DIS
LIN {X -144.015,Y 57.150,Z -121.781,A 90.000,B 90.000,C 0.000} C_DIS
LIN {X -144.015,Y 57.150,Z -114.232,A 90.000,B 90.000,C 0.000} C_DIS
LIN {X 144.015,Y 57.150,Z -114.232,A 90.000,B 90.000,C 0.000} C_DIS
LIN {X 144.015,Y 57.150,Z -106.683,A 90.000,B 90.000,C 0.000} C_DIS
LIN {X -144.015,Y 57.150,Z -106.683,A 90.000,B 90.000,C 0.000} C_DIS
LIN {X -144.015,Y 57.150,Z -99.134,A 90.000,B 90.000,C 0.000} C_DIS
LIN {X 144.015,Y 57.150,Z -99.134,A 90.000,B 90.000,C 0.000} C_DIS
LIN {X 144.015,Y 57.150,Z -91.586,A 90.000,B 90.000,C 0.000} C_DIS
LIN {X -144.015,Y 57.150,Z -91.586,A 90.000,B 90.000,C 0.000} C_DIS
LIN {X -144.015,Y 57.150,Z -84.037,A 90.000,B 90.000,C 0.000} C_DIS
LIN {X 144.015,Y 57.150,Z -84.037,A 90.000,B 90.000,C 0.000} C_DIS
LIN {X 144.015,Y 57.150,Z -76.488,A 90.000,B 90.000,C 0.000} C_DIS
LIN {X -144.015,Y 57.150,Z -76.488,A 90.000,B 90.000,C 0.000} C_DIS
LIN {X -144.015,Y 57.150,Z -68.939,A 90.000,B 90.000,C 0.000} C_DIS
LIN {X 144.015,Y 57.150,Z -68.939,A 90.000,B 90.000,C 0.000} C_DIS
LIN {X 144.015,Y 57.150,Z -61.390,A 90.000,B 90.000,C 0.000} C_DIS
LIN {X -144.015,Y 57.150,Z -61.390,A 90.000,B 90.000,C 0.000} C_DIS
LIN {X -144.015,Y 57.150,Z -53.842,A 90.000,B 90.000,C 0.000} C_DIS
LIN {X 144.015,Y 57.150,Z -53.842,A 90.000,B 90.000,C 0.000} C_DIS
LIN {X 144.015,Y 57.150,Z -46.293,A 90.000,B 90.000,C 0.000} C_DIS
LIN {X -144.015,Y 57.150,Z -46.293,A 90.000,B 90.000,C 0.000} C_DIS
LIN {X -144.015,Y 57.150,Z -38.744,A 90.000,B 90.000,C 0.000} C_DIS
LIN {X 144.015,Y 57.150,Z -38.744,A 90.000,B 90.000,C 0.000} C_DIS
LIN {X 144.015,Y 57.150,Z -31.195,A 90.000,B 90.000,C 0.000} C_DIS
LIN {X -144.015,Y 57.150,Z -31.195,A 90.000,B 90.000,C 0.000} C_DIS
LIN {X -144.015,Y 57.150,Z -23.646,A 90.000,B 90.000,C 0.000} C_DIS
LIN {X 144.015,Y 57.150,Z -23.646,A 90.000,B 90.000,C 0.000} C_DIS
LIN {X 144.015,Y 57.150,Z -16.098,A 90.000,B 90.000,C 0.000} C_DIS
LIN {X -144.015,Y 57.150,Z -16.098,A 90.000,B 90.000,C 0.000} C_DIS
LIN {X -144.015,Y 57.150,Z -8.549,A 90.000,B 90.000,C 0.000} C_DIS
LIN {X 144.015,Y 57.150,Z -8.549,A 90.000,B 90.000,C 0.000} C_DIS
LIN {X 144.015,Y 57.150,Z -1.000,A 90.000,B 90.000,C 0.000} C_DIS
LIN {X -144.015,Y 57.150,Z -1.000,A 90.000,B 90.000,C 0.000} C_DIS
LIN {X -145.015,Y 57.150,Z 0.000,A 90.000,B 90.000,C 0.000} C_DIS
LIN {X 145.015,Y 57.150,Z 0.000,A 90.000,B 90.000,C 0.000} C_DIS
LIN {X 145.015,Y 57.150,Z -243.561,A 90.000,B 90.000,C 0.000} C_DIS
LIN {X -145.015,Y 57.150,Z -243.561,A 90.000,B 90.000,C 0.000} C_DIS
LIN {X -145.015,Y 57.150,Z 0.000,A 90.000,B 90.000,C 0.000} C_DIS
LIN {X -145.015,Y 69.650,Z 0.000,A 90.000,B 90.000,C 0.000} C_DIS
LIN {X -145.015,Y 82.150,Z 0.000,A 90.000,B 90.000,C 0.000} C_DIS
LIN {X 144.015,Y 82.150,Z -242.561,A 90.000,B 90.000,C 0.000} C_DIS
LIN {X 144.015,Y 75.006,Z -242.561,A 90.000,B 90.000,C 0.000} C_DIS
LIN {X 144.015,Y 62.506,Z -242.561,A 90.000,B 90.000,C 0.000} C_DIS
LIN {X 144.015,Y 50.006,Z -242.561,A 90.000,B 90.000,C 0.000} C_DIS
LIN {X 34.059,Y 50.006,Z -242.561,A 90.000,B 90.000,C 0.000} C_DIS
LIN {X 35.200,Y 50.006,Z -242.066,A 90.000,B 90.000,C 0.000} C_DIS
LIN {X 36.314,Y 50.006,Z -241.512,A 90.000,B 90.000,C 0.000} C_DIS
LIN {X 37.398,Y 50.006,Z -240.901,A 90.000,B 90.000,C 0.000} C_DIS
LIN {X 38.448,Y 50.006,Z -240.234,A 90.000,B 90.000,C 0.000} C_DIS
LIN {X 39.463,Y 50.006,Z -239.514,A 90.000,B 90.000,C 0.000} C_DIS
LIN {X 40.438,Y 50.006,Z -238.741,A 90.000,B 90.000,C 0.000} C_DIS
LIN {X 41.372,Y 50.006,Z -237.919,A 90.000,B 90.000,C 0.000} C_DIS
LIN {X 42.262,Y 50.006,Z -237.050,A 90.000,B 90.000,C 0.000} C_DIS
LIN {X 44.273,Y 50.006,Z -235.012,A 90.000,B 90.000,C 0.000} C_DIS
LIN {X 144.015,Y 50.006,Z -235.012,A 90.000,B 90.000,C 0.000} C_DIS
LIN {X 144.015,Y 50.006,Z -227.464,A 90.000,B 90.000,C 0.000} C_DIS
LIN {X 49.291,Y 50.006,Z -227.464,A 90.000,B 90.000,C 0.000} C_DIS
LIN {X 49.985,Y 50.006,Z -226.001,A 90.000,B 90.000,C 0.000} C_DIS
LIN {X 50.621,Y 50.006,Z -224.513,A 90.000,B 90.000,C 0.000} C_DIS
LIN {X 51.200,Y 50.006,Z -223.000,A 90.000,B 90.000,C 0.000} C_DIS
LIN {X 51.720,Y 50.006,Z -221.467,A 90.000,B 90.000,C 0.000} C_DIS
LIN {X 52.180,Y 50.006,Z -219.915,A 90.000,B 90.000,C 0.000} C_DIS
LIN {X 144.015,Y 50.006,Z -219.915,A 90.000,B 90.000,C 0.000} C_DIS
LIN {X 144.015,Y 50.006,Z -212.366,A 90.000,B 90.000,C 0.000} C_DIS
LIN {X 54.147,Y 50.006,Z -212.366,A 90.000,B 90.000,C 0.000} C_DIS
LIN {X 54.682,Y 50.006,Z -210.400,A 90.000,B 90.000,C 0.000} C_DIS
LIN {X 55.225,Y 50.006,Z -208.436,A 90.000,B 90.000,C 0.000} C_DIS
LIN {X 55.444,Y 50.006,Z -207.731,A 90.000,B 90.000,C 0.000} C_DIS
LIN {X 55.617,Y 50.006,Z -207.014,A 90.000,B 90.000,C 0.000} C_DIS
LIN {X 55.744,Y 50.006,Z -206.288,A 90.000,B 90.000,C 0.000} C_DIS
LIN {X 55.823,Y 50.006,Z -205.554,A 90.000,B 90.000,C 0.000} C_DIS
LIN {X 55.855,Y 50.006,Z -204.817,A 90.000,B 90.000,C 0.000} C_DIS
LIN {X 144.015,Y 50.006,Z -204.817,A 90.000,B 90.000,C 0.000} C_DIS
LIN {X 144.015,Y 50.006,Z -197.269,A 90.000,B 90.000,C 0.000} C_DIS
LIN {X 55.372,Y 50.006,Z -197.269,A 90.000,B 90.000,C 0.000} C_DIS
LIN {X 55.371,Y 50.006,Z -196.761,A 90.000,B 90.000,C 0.000} C_DIS
LIN {X 55.264,Y 50.006,Z -195.954,A 90.000,B 90.000,C 0.000} C_DIS
LIN {X 55.095,Y 50.006,Z -195.159,A 90.000,B 90.000,C 0.000} C_DIS
LIN {X 54.866,Y 50.006,Z -194.378,A 90.000,B 90.000,C 0.000} C_DIS
LIN {X 54.576,Y 50.006,Z -193.618,A 90.000,B 90.000,C 0.000} C_DIS
LIN {X 54.229,Y 50.006,Z -192.882,A 90.000,B 90.000,C 0.000} C_DIS
LIN {X 53.826,Y 50.006,Z -192.175,A 90.000,B 90.000,C 0.000} C_DIS
LIN {X 53.369,Y 50.006,Z -191.502,A 90.000,B 90.000,C 0.000} C_DIS
LIN {X 52.862,Y 50.006,Z -190.865,A 90.000,B 90.000,C 0.000} C_DIS
LIN {X 52.307,Y 50.006,Z -190.270,A 90.000,B 90.000,C 0.000} C_DIS
LIN {X 51.708,Y 50.006,Z -189.720,A 90.000,B 90.000,C 0.000} C_DIS
LIN {X 144.015,Y 50.006,Z -189.720,A 90.000,B 90.000,C 0.000} C_DIS
LIN {X 144.015,Y 50.006,Z -182.171,A 90.000,B 90.000,C 0.000} C_DIS
LIN {X -144.015,Y 50.006,Z -182.171,A 90.000,B 90.000,C 0.000} C_DIS
LIN {X -144.015,Y 50.006,Z -174.622,A 90.000,B 90.000,C 0.000} C_DIS
LIN {X 144.015,Y 50.006,Z -174.622,A 90.000,B 90.000,C 0.000} C_DIS
LIN {X 144.015,Y 50.006,Z -167.073,A 90.000,B 90.000,C 0.000} C_DIS
LIN {X -144.015,Y 50.006,Z -167.073,A 90.000,B 90.000,C 0.000} C_DIS
LIN {X -144.015,Y 50.006,Z -159.525,A 90.000,B 90.000,C 0.000} C_DIS
LIN {X 144.015,Y 50.006,Z -159.525,A 90.000,B 90.000,C 0.000} C_DIS
LIN {X 144.015,Y 50.006,Z -151.976,A 90.000,B 90.000,C 0.000} C_DIS
LIN {X -144.015,Y 50.006,Z -151.976,A 90.000,B 90.000,C 0.000} C_DIS
LIN {X -144.015,Y 50.006,Z -144.427,A 90.000,B 90.000,C 0.000} C_DIS
LIN {X 0.837,Y 50.006,Z -144.427,A 90.000,B 90.000,C 0.000} C_DIS
LIN {X 0.136,Y 50.006,Z -144.011,A 90.000,B 90.000,C 0.000} C_DIS
LIN {X -0.540,Y 50.006,Z -143.555,A 90.000,B 90.000,C 0.000} C_DIS
LIN {X -1.189,Y 50.006,Z -143.061,A 90.000,B 90.000,C 0.000} C_DIS
LIN {X -1.808,Y 50.006,Z -142.530,A 90.000,B 90.000,C 0.000} C_DIS
LIN {X -2.396,Y 50.006,Z -141.965,A 90.000,B 90.000,C 0.000} C_DIS
LIN {X -3.002,Y 50.006,Z -141.460,A 90.000,B 90.000,C 0.000} C_DIS
LIN {X -3.569,Y 50.006,Z -140.910,A 90.000,B 90.000,C 0.000} C_DIS
LIN {X -4.093,Y 50.006,Z -140.320,A 90.000,B 90.000,C 0.000} C_DIS
LIN {X -4.571,Y 50.006,Z -139.692,A 90.000,B 90.000,C 0.000} C_DIS
LIN {X -5.000,Y 50.006,Z -139.030,A 90.000,B 90.000,C 0.000} C_DIS
LIN {X -5.379,Y 50.006,Z -138.338,A 90.000,B 90.000,C 0.000} C_DIS
LIN {X -5.705,Y 50.006,Z -137.619,A 90.000,B 90.000,C 0.000} C_DIS
LIN {X -5.976,Y 50.006,Z -136.878,A 90.000,B 90.000,C 0.000} C_DIS
LIN {X -144.015,Y 50.006,Z -136.878,A 90.000,B 90.000,C 0.000} C_DIS
LIN {X -144.015,Y 50.006,Z -129.329,A 90.000,B 90.000,C 0.000} C_DIS
LIN {X -6.782,Y 50.006,Z -129.329,A 90.000,B 90.000,C 0.000} C_DIS
LIN {X -6.694,Y 50.006,Z -128.830,A 90.000,B 90.000,C 0.000} C_DIS
LIN {X -6.588,Y 50.006,Z -128.335,A 90.000,B 90.000,C 0.000} C_DIS
LIN {X -6.310,Y 50.006,Z -127.531,A 90.000,B 90.000,C 0.000} C_DIS
LIN {X -5.977,Y 50.006,Z -126.747,A 90.000,B 90.000,C 0.000} C_DIS
LIN {X -5.591,Y 50.006,Z -125.988,A 90.000,B 90.000,C 0.000} C_DIS
LIN {X -5.154,Y 50.006,Z -125.257,A 90.000,B 90.000,C 0.000} C_DIS
LIN {X -4.668,Y 50.006,Z -124.558,A 90.000,B 90.000,C 0.000} C_DIS
LIN {X -4.136,Y 50.006,Z -123.894,A 90.000,B 90.000,C 0.000} C_DIS
LIN {X -3.611,Y 50.006,Z -123.164,A 90.000,B 90.000,C 0.000} C_DIS
LIN {X -3.054,Y 50.006,Z -122.459,A 90.000,B 90.000,C 0.000} C_DIS
LIN {X -2.464,Y 50.006,Z -121.781,A 90.000,B 90.000,C 0.000} C_DIS
LIN {X -144.015,Y 50.006,Z -121.781,A 90.000,B 90.000,C 0.000} C_DIS
LIN {X -144.015,Y 50.006,Z -114.232,A 90.000,B 90.000,C 0.000} C_DIS
LIN {X 144.015,Y 50.006,Z -114.232,A 90.000,B 90.000,C 0.000} C_DIS
LIN {X 144.015,Y 50.006,Z -106.683,A 90.000,B 90.000,C 0.000} C_DIS
LIN {X -144.015,Y 50.006,Z -106.683,A 90.000,B 90.000,C 0.000} C_DIS
LIN {X -144.015,Y 50.006,Z -99.134,A 90.000,B 90.000,C 0.000} C_DIS
LIN {X 144.015,Y 50.006,Z -99.134,A 90.000,B 90.000,C 0.000} C_DIS
LIN {X 144.015,Y 50.006,Z -91.586,A 90.000,B 90.000,C 0.000} C_DIS
LIN {X -144.015,Y 50.006,Z -91.586,A 90.000,B 90.000,C 0.000} C_DIS
LIN {X -144.015,Y 50.006,Z -84.037,A 90.000,B 90.000,C 0.000} C_DIS
LIN {X 144.015,Y 50.006,Z -84.037,A 90.000,B 90.000,C 0.000} C_DIS
LIN {X 144.015,Y 50.006,Z -76.488,A 90.000,B 90.000,C 0.000} C_DIS
LIN {X 102.694,Y 50.006,Z -76.488,A 90.000,B 90.000,C 0.000} C_DIS
LIN {X 103.530,Y 50.006,Z -75.880,A 90.000,B 90.000,C 0.000} C_DIS
LIN {X 104.333,Y 50.006,Z -75.229,A 90.000,B 90.000,C 0.000} C_DIS
LIN {X 105.101,Y 50.006,Z -74.538,A 90.000,B 90.000,C 0.000} C_DIS
LIN {X 105.832,Y 50.006,Z -73.807,A 90.000,B 90.000,C 0.000} C_DIS
LIN {X 106.524,Y 50.006,Z -73.039,A 90.000,B 90.000,C 0.000} C_DIS
LIN {X 107.347,Y 50.006,Z -72.058,A 90.000,B 90.000,C 0.000} C_DIS
LIN {X 108.134,Y 50.006,Z -71.046,A 90.000,B 90.000,C 0.000} C_DIS
LIN {X 108.882,Y 50.006,Z -70.006,A 90.000,B 90.000,C 0.000} C_DIS
LIN {X 109.590,Y 50.006,Z -68.939,A 90.000,B 90.000,C 0.000} C_DIS
LIN {X 144.015,Y 50.006,Z -68.939,A 90.000,B 90.000,C 0.000} C_DIS
LIN {X 144.015,Y 50.006,Z -61.390,A 90.000,B 90.000,C 0.000} C_DIS
LIN {X 113.192,Y 50.006,Z -61.390,A 90.000,B 90.000,C 0.000} C_DIS
LIN {X 113.580,Y 50.006,Z -60.153,A 90.000,B 90.000,C 0.000} C_DIS
LIN {X 113.922,Y 50.006,Z -58.901,A 90.000,B 90.000,C 0.000} C_DIS
LIN {X 114.215,Y 50.006,Z -57.638,A 90.000,B 90.000,C 0.000} C_DIS
LIN {X 114.462,Y 50.006,Z -56.365,A 90.000,B 90.000,C 0.000} C_DIS
LIN {X 114.561,Y 50.006,Z -55.102,A 90.000,B 90.000,C 0.000} C_DIS
LIN {X 114.692,Y 50.006,Z -53.842,A 90.000,B 90.000,C 0.000} C_DIS
LIN {X 144.015,Y 50.006,Z -53.842,A 90.000,B 90.000,C 0.000} C_DIS
LIN {X 144.015,Y 50.006,Z -46.293,A 90.000,B 90.000,C 0.000} C_DIS
LIN {X 115.066,Y 50.006,Z -46.293,A 90.000,B 90.000,C 0.000} C_DIS
LIN {X 114.879,Y 50.006,Z -45.406,A 90.000,B 90.000,C 0.000} C_DIS
LIN {X 114.625,Y 50.006,Z -44.536,A 90.000,B 90.000,C 0.000} C_DIS
LIN {X 114.306,Y 50.006,Z -43.687,A 90.000,B 90.000,C 0.000} C_DIS
LIN {X 113.924,Y 50.006,Z -42.865,A 90.000,B 90.000,C 0.000} C_DIS
LIN {X 113.480,Y 50.006,Z -42.075,A 90.000,B 90.000,C 0.000} C_DIS
LIN {X 112.978,Y 50.006,Z -41.320,A 90.000,B 90.000,C 0.000} C_DIS
LIN {X 112.419,Y 50.006,Z -40.606,A 90.000,B 90.000,C 0.000} C_DIS
LIN {X 111.809,Y 50.006,Z -39.936,A 90.000,B 90.000,C 0.000} C_DIS
LIN {X 111.149,Y 50.006,Z -39.314,A 90.000,B 90.000,C 0.000} C_DIS
LIN {X 110.444,Y 50.006,Z -38.744,A 90.000,B 90.000,C 0.000} C_DIS
LIN {X 144.015,Y 50.006,Z -38.744,A 90.000,B 90.000,C 0.000} C_DIS
LIN {X 144.015,Y 50.006,Z -31.195,A 90.000,B 90.000,C 0.000} C_DIS
LIN {X -144.015,Y 50.006,Z -31.195,A 90.000,B 90.000,C 0.000} C_DIS
LIN {X -144.015,Y 50.006,Z -23.646,A 90.000,B 90.000,C 0.000} C_DIS
LIN {X 144.015,Y 50.006,Z -23.646,A 90.000,B 90.000,C 0.000} C_DIS
LIN {X 144.015,Y 50.006,Z -16.098,A 90.000,B 90.000,C 0.000} C_DIS
LIN {X -144.015,Y 50.006,Z -16.098,A 90.000,B 90.000,C 0.000} C_DIS
LIN {X -144.015,Y 50.006,Z -8.549,A 90.000,B 90.000,C 0.000} C_DIS
LIN {X 144.015,Y 50.006,Z -8.549,A 90.000,B 90.000,C 0.000} C_DIS
LIN {X 144.015,Y 50.006,Z -1.000,A 90.000,B 90.000,C 0.000} C_DIS
LIN {X -144.015,Y 50.006,Z -1.000,A 90.000,B 90.000,C 0.000} C_DIS
LIN {X -144.015,Y 50.006,Z -38.744,A 90.000,B 90.000,C 0.000} C_DIS
LIN {X 95.847,Y 50.006,Z -38.744,A 90.000,B 90.000,C 0.000} C_DIS
LIN {X 95.119,Y 50.006,Z -39.194,A 90.000,B 90.000,C 0.000} C_DIS
LIN {X 94.407,Y 50.006,Z -39.671,A 90.000,B 90.000,C 0.000} C_DIS
LIN {X 93.713,Y 50.006,Z -40.172,A 90.000,B 90.000,C 0.000} C_DIS
LIN {X 91.733,Y 50.006,Z -41.964,A 90.000,B 90.000,C 0.000} C_DIS
LIN {X 89.723,Y 50.006,Z -43.723,A 90.000,B 90.000,C 0.000} C_DIS
LIN {X 87.685,Y 50.006,Z -45.449,A 90.000,B 90.000,C 0.000} C_DIS
LIN {X 87.149,Y 50.006,Z -45.868,A 90.000,B 90.000,C 0.000} C_DIS
LIN {X 86.618,Y 50.006,Z -46.293,A 90.000,B 90.000,C 0.000} C_DIS
LIN {X -144.015,Y 50.006,Z -46.293,A 90.000,B 90.000,C 0.000} C_DIS
LIN {X -144.015,Y 50.006,Z -53.842,A 90.000,B 90.000,C 0.000} C_DIS
LIN {X 78.955,Y 50.006,Z -53.842,A 90.000,B 90.000,C 0.000} C_DIS
LIN {X 78.303,Y 50.006,Z -54.681,A 90.000,B 90.000,C 0.000} C_DIS
LIN {X 77.704,Y 50.006,Z -55.559,A 90.000,B 90.000,C 0.000} C_DIS
LIN {X 77.160,Y 50.006,Z -56.472,A 90.000,B 90.000,C 0.000} C_DIS
LIN {X 76.673,Y 50.006,Z -57.416,A 90.000,B 90.000,C 0.000} C_DIS
LIN {X 76.244,Y 50.006,Z -58.388,A 90.000,B 90.000,C 0.000} C_DIS
LIN {X 75.875,Y 50.006,Z -59.385,A 90.000,B 90.000,C 0.000} C_DIS
LIN {X 75.568,Y 50.006,Z -60.402,A 90.000,B 90.000,C 0.000} C_DIS
LIN {X 75.431,Y 50.006,Z -60.894,A 90.000,B 90.000,C 0.000} C_DIS
LIN {X 75.310,Y 50.006,Z -61.390,A 90.000,B 90.000,C 0.000} C_DIS
LIN {X -144.015,Y 50.006,Z -61.390,A 90.000,B 90.000,C 0.000} C_DIS
LIN {X -144.015,Y 50.006,Z -68.939,A 90.000,B 90.000,C 0.000} C_DIS
LIN {X 75.650,Y 50.006,Z -68.939,A 90.000,B 90.000,C 0.000} C_DIS
LIN {X 75.973,Y 50.006,Z -69.843,A 90.000,B 90.000,C 0.000} C_DIS
LIN {X 76.355,Y 50.006,Z -70.724,A 90.000,B 90.000,C 0.000} C_DIS
LIN {X 76.794,Y 50.006,Z -71.577,A 90.000,B 90.000,C 0.000} C_DIS
LIN {X 77.290,Y 50.006,Z -72.399,A 90.000,B 90.000,C 0.000} C_DIS
LIN {X 77.838,Y 50.006,Z -73.187,A 90.000,B 90.000,C 0.000} C_DIS
LIN {X 78.438,Y 50.006,Z -73.936,A 90.000,B 90.000,C 0.000} C_DIS
LIN {X 79.087,Y 50.006,Z -74.644,A 90.000,B 90.000,C 0.000} C_DIS
LIN {X 79.781,Y 50.006,Z -75.307,A 90.000,B 90.000,C 0.000} C_DIS
LIN {X 80.517,Y 50.006,Z -75.923,A 90.000,B 90.000,C 0.000} C_DIS
LIN {X 81.293,Y 50.006,Z -76.488,A 90.000,B 90.000,C 0.000} C_DIS
LIN {X -144.015,Y 50.006,Z -76.488,A 90.000,B 90.000,C 0.000} C_DIS
LIN {X -144.015,Y 50.006,Z -189.720,A 90.000,B 90.000,C 0.000} C_DIS
LIN {X 36.184,Y 50.006,Z -189.720,A 90.000,B 90.000,C 0.000} C_DIS
LIN {X 35.390,Y 50.006,Z -190.142,A 90.000,B 90.000,C 0.000} C_DIS
LIN {X 34.631,Y 50.006,Z -190.625,A 90.000,B 90.000,C 0.000} C_DIS
LIN {X 33.913,Y 50.006,Z -191.165,A 90.000,B 90.000,C 0.000} C_DIS
LIN {X 33.238,Y 50.006,Z -191.759,A 90.000,B 90.000,C 0.000} C_DIS
LIN {X 32.612,Y 50.006,Z -192.405,A 90.000,B 90.000,C 0.000} C_DIS
LIN {X 32.038,Y 50.006,Z -193.097,A 90.000,B 90.000,C 0.000} C_DIS
LIN {X 31.519,Y 50.006,Z -193.831,A 90.000,B 90.000,C 0.000} C_DIS
LIN {X 31.060,Y 50.006,Z -194.604,A 90.000,B 90.000,C 0.000} C_DIS
LIN {X 30.390,Y 50.006,Z -195.469,A 90.000,B 90.000,C 0.000} C_DIS
LIN {X 29.750,Y 50.006,Z -196.358,A 90.000,B 90.000,C 0.000} C_DIS
LIN {X 29.143,Y 50.006,Z -197.269,A 90.000,B 90.000,C 0.000} C_DIS
LIN {X -144.015,Y 50.006,Z -197.269,A 90.000,B 90.000,C 0.000} C_DIS
LIN {X -144.015,Y 50.006,Z -204.817,A 90.000,B 90.000,C 0.000} C_DIS
LIN {X 24.426,Y 50.006,Z -204.817,A 90.000,B 90.000,C 0.000} C_DIS
LIN {X 22.929,Y 50.006,Z -207.306,A 90.000,B 90.000,C 0.000} C_DIS
LIN {X 21.479,Y 50.006,Z -209.823,A 90.000,B 90.000,C 0.000} C_DIS
LIN {X 20.076,Y 50.006,Z -212.366,A 90.000,B 90.000,C 0.000} C_DIS
LIN {X -144.015,Y 50.006,Z -212.366,A 90.000,B 90.000,C 0.000} C_DIS
LIN {X -144.015,Y 50.006,Z -219.915,A 90.000,B 90.000,C 0.000} C_DIS
LIN {X 16.295,Y 50.006,Z -219.915,A 90.000,B 90.000,C 0.000} C_DIS
LIN {X 15.879,Y 50.006,Z -221.001,A 90.000,B 90.000,C 0.000} C_DIS
LIN {X 15.509,Y 50.006,Z -222.103,A 90.000,B 90.000,C 0.000} C_DIS
LIN {X 15.186,Y 50.006,Z -223.220,A 90.000,B 90.000,C 0.000} C_DIS
LIN {X 14.911,Y 50.006,Z -224.350,A 90.000,B 90.000,C 0.000} C_DIS
LIN {X 14.683,Y 50.006,Z -225.490,A 90.000,B 90.000,C 0.000} C_DIS
LIN {X 14.503,Y 50.006,Z -226.639,A 90.000,B 90.000,C 0.000} C_DIS
LIN {X 14.494,Y 50.006,Z -227.464,A 90.000,B 90.000,C 0.000} C_DIS
LIN {X -144.015,Y 50.006,Z -227.464,A 90.000,B 90.000,C 0.000} C_DIS
LIN {X -144.015,Y 50.006,Z -235.012,A 90.000,B 90.000,C 0.000} C_DIS
LIN {X -56.979,Y 50.006,Z -235.012,A 90.000,B 90.000,C 0.000} C_DIS
LIN {X -58.737,Y 50.006,Z -235.637,A 90.000,B 90.000,C 0.000} C_DIS
LIN {X -60.486,Y 50.006,Z -236.289,A 90.000,B 90.000,C 0.000} C_DIS
LIN {X -63.186,Y 50.006,Z -237.439,A 90.000,B 90.000,C 0.000} C_DIS
LIN {X -65.864,Y 50.006,Z -238.642,A 90.000,B 90.000,C 0.000} C_DIS
LIN {X -68.517,Y 50.006,Z -239.897,A 90.000,B 90.000,C 0.000} C_DIS
LIN {X -71.146,Y 50.006,Z -241.204,A 90.000,B 90.000,C 0.000} C_DIS
LIN {X -73.748,Y 50.006,Z -242.561,A 90.000,B 90.000,C 0.000} C_DIS
LIN {X -144.015,Y 50.006,Z -242.561,A 90.000,B 90.000,C 0.000} C_DIS
LIN {X -62.734,Y 50.006,Z -237.242,A 90.000,B 90.000,C 0.000} C_DIS
LIN {X -61.612,Y 50.006,Z -236.761,A 90.000,B 90.000,C 0.000} C_DIS
LIN {X -60.486,Y 50.006,Z -236.289,A 90.000,B 90.000,C 0.000} C_DIS
LIN {X -58.137,Y 50.006,Z -235.420,A 90.000,B 90.000,C 0.000} C_DIS
LIN {X -55.770,Y 50.006,Z -234.600,A 90.000,B 90.000,C 0.000} C_DIS
LIN {X -53.387,Y 50.006,Z -233.829,A 90.000,B 90.000,C 0.000} C_DIS
LIN {X -50.988,Y 50.006,Z -233.108,A 90.000,B 90.000,C 0.000} C_DIS
LIN {X -49.470,Y 50.006,Z -232.745,A 90.000,B 90.000,C 0.000} C_DIS
LIN {X -47.939,Y 50.006,Z -232.440,A 90.000,B 90.000,C 0.000} C_DIS
LIN {X -46.397,Y 50.006,Z -232.192,A 90.000,B 90.000,C 0.000} C_DIS
LIN {X -44.848,Y 50.006,Z -232.001,A 90.000,B 90.000,C 0.000} C_DIS
LIN {X -43.292,Y 50.006,Z -231.869,A 90.000,B 90.000,C 0.000} C_DIS
LIN {X -41.733,Y 50.006,Z -231.795,A 90.000,B 90.000,C 0.000} C_DIS
LIN {X -40.172,Y 50.006,Z -231.780,A 90.000,B 90.000,C 0.000} C_DIS
LIN {X -39.001,Y 50.006,Z -231.838,A 90.000,B 90.000,C 0.000} C_DIS
LIN {X -37.834,Y 50.006,Z -231.946,A 90.000,B 90.000,C 0.000} C_DIS
LIN {X -36.672,Y 50.006,Z -232.103,A 90.000,B 90.000,C 0.000} C_DIS
LIN {X -35.518,Y 50.006,Z -232.311,A 90.000,B 90.000,C 0.000} C_DIS
LIN {X -34.374,Y 50.006,Z -232.567,A 90.000,B 90.000,C 0.000} C_DIS
LIN {X -33.242,Y 50.006,Z -232.871,A 90.000,B 90.000,C 0.000} C_DIS
LIN {X -32.124,Y 50.006,Z -233.224,A 90.000,B 90.000,C 0.000} C_DIS
LIN {X -31.237,Y 50.006,Z -233.629,A 90.000,B 90.000,C 0.000} C_DIS
LIN {X -30.363,Y 50.006,Z -234.062,A 90.000,B 90.000,C 0.000} C_DIS
LIN {X -29.503,Y 50.006,Z -234.523,A 90.000,B 90.000,C 0.000} C_DIS
LIN {X -28.659,Y 50.006,Z -235.012,A 90.000,B 90.000,C 0.000} C_DIS
LIN {X 15.345,Y 50.006,Z -235.012,A 90.000,B 90.000,C 0.000} C_DIS
LIN {X 15.610,Y 50.006,Z -235.821,A 90.000,B 90.000,C 0.000} C_DIS
LIN {X 15.940,Y 50.006,Z -236.606,A 90.000,B 90.000,C 0.000} C_DIS
LIN {X 16.332,Y 50.006,Z -237.362,A 90.000,B 90.000,C 0.000} C_DIS
LIN {X 16.784,Y 50.006,Z -238.084,A 90.000,B 90.000,C 0.000} C_DIS
LIN {X 17.293,Y 50.006,Z -238.767,A 90.000,B 90.000,C 0.000} C_DIS
LIN {X 17.855,Y 50.006,Z -239.406,A 90.000,B 90.000,C 0.000} C_DIS
LIN {X 18.468,Y 50.006,Z -239.998,A 90.000,B 90.000,C 0.000} C_DIS
LIN {X 19.126,Y 50.006,Z -240.538,A 90.000,B 90.000,C 0.000} C_DIS
LIN {X 19.842,Y 50.006,Z -240.984,A 90.000,B 90.000,C 0.000} C_DIS
LIN {X 20.582,Y 50.006,Z -241.388,A 90.000,B 90.000,C 0.000} C_DIS
LIN {X 21.344,Y 50.006,Z -241.749,A 90.000,B 90.000,C 0.000} C_DIS
LIN {X 22.125,Y 50.006,Z -242.066,A 90.000,B 90.000,C 0.000} C_DIS
LIN {X 22.924,Y 50.006,Z -242.337,A 90.000,B 90.000,C 0.000} C_DIS
LIN {X 23.737,Y 50.006,Z -242.561,A 90.000,B 90.000,C 0.000} C_DIS
LIN {X -21.157,Y 50.006,Z -242.561,A 90.000,B 90.000,C 0.000} C_DIS
LIN {X 17.180,Y 50.006,Z -144.427,A 90.000,B 90.000,C 0.000} C_DIS
LIN {X 144.015,Y 50.006,Z -144.427,A 90.000,B 90.000,C 0.000} C_DIS
LIN {X 144.015,Y 50.006,Z -136.878,A 90.000,B 90.000,C 0.000} C_DIS
LIN {X 26.237,Y 50.006,Z -136.878,A 90.000,B 90.000,C 0.000} C_DIS
LIN {X 26.714,Y 50.006,Z -136.011,A 90.000,B 90.000,C 0.000} C_DIS
LIN {X 27.130,Y 50.006,Z -135.114,A 90.000,B 90.000,C 0.000} C_DIS
LIN {X 27.484,Y 50.006,Z -134.190,A 90.000,B 90.000,C 0.000} C_DIS
LIN {X 27.773,Y 50.006,Z -133.244,A 90.000,B 90.000,C 0.000} C_DIS
LIN {X 27.997,Y 50.006,Z -132.280,A 90.000,B 90.000,C 0.000} C_DIS
LIN {X 28.153,Y 50.006,Z -131.303,A 90.000,B 90.000,C 0.000} C_DIS
LIN {X 28.242,Y 50.006,Z -130.318,A 90.000,B 90.000,C 0.000} C_DIS
LIN {X 28.264,Y 50.006,Z -129.329,A 90.000,B 90.000,C 0.000} C_DIS
LIN {X 144.015,Y 50.006,Z -129.329,A 90.000,B 90.000,C 0.000} C_DIS
LIN {X 144.015,Y 50.006,Z -121.781,A 90.000,B 90.000,C 0.000} C_DIS
LIN {X 26.111,Y 50.006,Z -121.781,A 90.000,B 90.000,C 0.000} C_DIS
LIN {X 25.941,Y 50.006,Z -123.710,A 90.000,B 90.000,C 0.000} C_DIS
LIN {X 25.594,Y 50.006,Z -122.929,A 90.000,B 90.000,C 0.000} C_DIS
LIN {X 25.186,Y 50.006,Z -122.179,A 90.000,B 90.000,C 0.000} C_DIS
LIN {X 24.718,Y 50.006,Z -121.465,A 90.000,B 90.000,C 0.000} C_DIS
LIN {X 24.194,Y 50.006,Z -120.790,A 90.000,B 90.000,C 0.000} C_DIS
LIN {X 23.617,Y 50.006,Z -120.160,A 90.000,B 90.000,C 0.000} C_DIS
LIN {X 22.991,Y 50.006,Z -119.579,A 90.000,B 90.000,C 0.000} C_DIS
LIN {X 22.320,Y 50.006,Z -119.050,A 90.000,B 90.000,C 0.000} C_DIS
LIN {X 21.609,Y 50.006,Z -118.577,A 90.000,B 90.000,C 0.000} C_DIS
LIN {X 20.862,Y 50.006,Z -118.163,A 90.000,B 90.000,C 0.000} C_DIS
LIN {X 19.415,Y 50.006,Z -117.625,A 90.000,B 90.000,C 0.000} C_DIS
LIN {X 17.948,Y 50.006,Z -117.141,A 90.000,B 90.000,C 0.000} C_DIS
LIN {X 16.464,Y 50.006,Z -116.714,A 90.000,B 90.000,C 0.000} C_DIS
LIN {X 14.965,Y 50.006,Z -116.342,A 90.000,B 90.000,C 0.000} C_DIS
LIN {X 13.767,Y 50.006,Z -116.304,A 90.000,B 90.000,C 0.000} C_DIS
LIN {X 12.569,Y 50.006,Z -116.320,A 90.000,B 90.000,C 0.000} C_DIS
LIN {X 11.373,Y 50.006,Z -116.392,A 90.000,B 90.000,C 0.000} C_DIS
LIN {X 10.181,Y 50.006,Z -116.518,A 90.000,B 90.000,C 0.000} C_DIS
LIN {X 8.997,Y 50.006,Z -116.699,A 90.000,B 90.000,C 0.000} C_DIS
LIN {X 7.822,Y 50.006,Z -116.934,A 90.000,B 90.000,C 0.000} C_DIS
LIN {X 6.725,Y 50.006,Z -117.273,A 90.000,B 90.000,C 0.000} C_DIS
LIN {X 5.644,Y 50.006,Z -117.662,A 90.000,B 90.000,C 0.000} C_DIS
LIN {X 4.583,Y 50.006,Z -118.101,A 90.000,B 90.000,C 0.000} C_DIS
LIN {X 3.543,Y 50.006,Z -118.587,A 90.000,B 90.000,C 0.000} C_DIS
LIN {X 2.526,Y 50.006,Z -119.122,A 90.000,B 90.000,C 0.000} C_DIS
LIN {X 1.535,Y 50.006,Z -119.702,A 90.000,B 90.000,C 0.000} C_DIS
LIN {X 0.572,Y 50.006,Z -120.327,A 90.000,B 90.000,C 0.000} C_DIS
LIN {X -0.168,Y 50.006,Z -120.935,A 90.000,B 90.000,C 0.000} C_DIS
LIN {X -0.875,Y 50.006,Z -121.581,A 90.000,B 90.000,C 0.000} C_DIS
LIN {X -1.548,Y 50.006,Z -122.263,A 90.000,B 90.000,C 0.000} C_DIS
LIN {X -2.185,Y 50.006,Z -122.978,A 90.000,B 90.000,C 0.000} C_DIS
LIN {X -2.783,Y 50.006,Z -123.726,A 90.000,B 90.000,C 0.000} C_DIS
LIN {X -3.342,Y 50.006,Z -124.504,A 90.000,B 90.000,C 0.000} C_DIS
LIN {X -3.837,Y 50.006,Z -125.115,A 90.000,B 90.000,C 0.000} C_DIS
LIN {X -4.288,Y 50.006,Z -125.759,A 90.000,B 90.000,C 0.000} C_DIS
LIN {X -4.694,Y 50.006,Z -126.432,A 90.000,B 90.000,C 0.000} C_DIS
LIN {X -5.053,Y 50.006,Z -127.132,A 90.000,B 90.000,C 0.000} C_DIS
LIN {X -5.363,Y 50.006,Z -127.855,A 90.000,B 90.000,C 0.000} C_DIS
LIN {X -5.622,Y 50.006,Z -128.597,A 90.000,B 90.000,C 0.000} C_DIS
LIN {X -5.789,Y 50.006,Z -129.454,A 90.000,B 90.000,C 0.000} C_DIS
LIN {X -5.898,Y 50.006,Z -130.320,A 90.000,B 90.000,C 0.000} C_DIS
LIN {X -5.947,Y 50.006,Z -131.191,A 90.000,B 90.000,C 0.000} C_DIS
LIN {X -5.936,Y 50.006,Z -132.064,A 90.000,B 90.000,C 0.000} C_DIS
LIN {X -5.867,Y 50.006,Z -132.933,A 90.000,B 90.000,C 0.000} C_DIS
LIN {X -5.738,Y 50.006,Z -133.797,A 90.000,B 90.000,C 0.000} C_DIS
LIN {X -5.551,Y 50.006,Z -134.649,A 90.000,B 90.000,C 0.000} C_DIS
LIN {X -5.307,Y 50.006,Z -135.487,A 90.000,B 90.000,C 0.000} C_DIS
LIN {X -5.128,Y 50.006,Z -136.233,A 90.000,B 90.000,C 0.000} C_DIS
LIN {X -4.889,Y 50.006,Z -136.961,A 90.000,B 90.000,C 0.000} C_DIS
LIN {X -4.592,Y 50.006,Z -137.668,A 90.000,B 90.000,C 0.000} C_DIS
LIN {X -4.240,Y 50.006,Z -138.349,A 90.000,B 90.000,C 0.000} C_DIS
LIN {X -3.834,Y 50.006,Z -139.000,A 90.000,B 90.000,C 0.000} C_DIS
LIN {X -3.377,Y 50.006,Z -139.616,A 90.000,B 90.000,C 0.000} C_DIS
LIN {X -2.871,Y 50.006,Z -140.192,A 90.000,B 90.000,C 0.000} C_DIS
LIN {X -2.321,Y 50.006,Z -140.727,A 90.000,B 90.000,C 0.000} C_DIS
LIN {X -1.730,Y 50.006,Z -141.215,A 90.000,B 90.000,C 0.000} C_DIS
LIN {X -1.055,Y 50.006,Z -141.862,A 90.000,B 90.000,C 0.000} C_DIS
LIN {X -0.336,Y 50.006,Z -142.460,A 90.000,B 90.000,C 0.000} C_DIS
LIN {X 0.423,Y 50.006,Z -143.005,A 90.000,B 90.000,C 0.000} C_DIS
LIN {X 1.220,Y 50.006,Z -143.495,A 90.000,B 90.000,C 0.000} C_DIS
LIN {X 2.049,Y 50.006,Z -143.927,A 90.000,B 90.000,C 0.000} C_DIS
LIN {X 2.906,Y 50.006,Z -144.300,A 90.000,B 90.000,C 0.000} C_DIS
LIN {X 3.788,Y 50.006,Z -144.610,A 90.000,B 90.000,C 0.000} C_DIS
LIN {X 4.690,Y 50.006,Z -144.858,A 90.000,B 90.000,C 0.000} C_DIS
LIN {X 5.999,Y 50.006,Z -144.976,A 90.000,B 90.000,C 0.000} C_DIS
LIN {X 7.312,Y 50.006,Z -145.040,A 90.000,B 90.000,C 0.000} C_DIS
LIN {X 8.626,Y 50.006,Z -145.051,A 90.000,B 90.000,C 0.000} C_DIS
LIN {X 9.940,Y 50.006,Z -145.008,A 90.000,B 90.000,C 0.000} C_DIS
LIN {X 11.251,Y 50.006,Z -144.912,A 90.000,B 90.000,C 0.000} C_DIS
LIN {X 12.557,Y 50.006,Z -144.762,A 90.000,B 90.000,C 0.000} C_DIS
LIN {X 14.156,Y 50.006,Z -144.316,A 90.000,B 90.000,C 0.000} C_DIS
LIN {X 15.746,Y 50.006,Z -143.837,A 90.000,B 90.000,C 0.000} C_DIS
LIN {X 17.325,Y 50.006,Z -143.325,A 90.000,B 90.000,C 0.000} C_DIS
LIN {X 18.171,Y 50.006,Z -142.987,A 90.000,B 90.000,C 0.000} C_DIS
LIN {X 18.994,Y 50.006,Z -142.594,A 90.000,B 90.000,C 0.000} C_DIS
LIN {X 19.790,Y 50.006,Z -142.148,A 90.000,B 90.000,C 0.000} C_DIS
LIN {X 20.554,Y 50.006,Z -141.652,A 90.000,B 90.000,C 0.000} C_DIS
LIN {X 21.285,Y 50.006,Z -141.107,A 90.000,B 90.000,C 0.000} C_DIS
LIN {X 21.979,Y 50.006,Z -140.516,A 90.000,B 90.000,C 0.000} C_DIS
LIN {X 22.632,Y 50.006,Z -139.880,A 90.000,B 90.000,C 0.000} C_DIS
LIN {X 23.243,Y 50.006,Z -139.204,A 90.000,B 90.000,C 0.000} C_DIS
LIN {X 23.809,Y 50.006,Z -138.489,A 90.000,B 90.000,C 0.000} C_DIS
LIN {X 24.445,Y 50.006,Z -137.731,A 90.000,B 90.000,C 0.000} C_DIS
LIN {X 25.024,Y 50.006,Z -136.928,A 90.000,B 90.000,C 0.000} C_DIS
LIN {X 25.541,Y 50.006,Z -136.084,A 90.000,B 90.000,C 0.000} C_DIS
LIN {X 25.995,Y 50.006,Z -135.204,A 90.000,B 90.000,C 0.000} C_DIS
LIN {X 26.382,Y 50.006,Z -134.293,A 90.000,B 90.000,C 0.000} C_DIS
LIN {X 26.701,Y 50.006,Z -133.356,A 90.000,B 90.000,C 0.000} C_DIS
LIN {X 26.950,Y 50.006,Z -132.398,A 90.000,B 90.000,C 0.000} C_DIS
LIN {X 27.128,Y 50.006,Z -131.425,A 90.000,B 90.000,C 0.000} C_DIS
LIN {X 27.232,Y 50.006,Z -130.440,A 90.000,B 90.000,C 0.000} C_DIS
LIN {X 27.264,Y 50.006,Z -129.451,A 90.000,B 90.000,C 0.000} C_DIS
LIN {X 27.223,Y 50.006,Z -128.462,A 90.000,B 90.000,C 0.000} C_DIS
LIN {X 27.109,Y 50.006,Z -127.479,A 90.000,B 90.000,C 0.000} C_DIS
LIN {X 26.922,Y 50.006,Z -126.507,A 90.000,B 90.000,C 0.000} C_DIS
LIN {X 26.664,Y 50.006,Z -125.551,A 90.000,B 90.000,C 0.000} C_DIS
LIN {X 26.336,Y 50.006,Z -124.618,A 90.000,B 90.000,C 0.000} C_DIS
LIN {X 25.941,Y 50.006,Z -123.710,A 90.000,B 90.000,C 0.000} C_DIS
LIN {X 26.287,Y 50.006,Z -124.492,A 90.000,B 90.000,C 0.000} C_DIS
LIN {X 26.583,Y 50.006,Z -125.294,A 90.000,B 90.000,C 0.000} C_DIS
LIN {X 26.826,Y 50.006,Z -126.114,A 90.000,B 90.000,C 0.000} C_DIS
LIN {X 27.017,Y 50.006,Z -126.947,A 90.000,B 90.000,C 0.000} C_DIS
LIN {X 27.154,Y 50.006,Z -127.791,A 90.000,B 90.000,C 0.000} C_DIS
LIN {X 45.115,Y 50.006,Z -188.217,A 90.000,B 90.000,C 0.000} C_DIS
LIN {X 44.102,Y 50.006,Z -188.315,A 90.000,B 90.000,C 0.000} C_DIS
LIN {X 43.098,Y 50.006,Z -188.477,A 90.000,B 90.000,C 0.000} C_DIS
LIN {X 42.106,Y 50.006,Z -188.703,A 90.000,B 90.000,C 0.000} C_DIS
LIN {X 41.130,Y 50.006,Z -188.993,A 90.000,B 90.000,C 0.000} C_DIS
LIN {X 40.175,Y 50.006,Z -189.344,A 90.000,B 90.000,C 0.000} C_DIS
LIN {X 39.245,Y 50.006,Z -189.756,A 90.000,B 90.000,C 0.000} C_DIS
LIN {X 38.410,Y 50.006,Z -189.949,A 90.000,B 90.000,C 0.000} C_DIS
LIN {X 37.593,Y 50.006,Z -190.210,A 90.000,B 90.000,C 0.000} C_DIS
LIN {X 36.800,Y 50.006,Z -190.536,A 90.000,B 90.000,C 0.000} C_DIS
LIN {X 36.036,Y 50.006,Z -190.925,A 90.000,B 90.000,C 0.000} C_DIS
LIN {X 35.306,Y 50.006,Z -191.375,A 90.000,B 90.000,C 0.000} C_DIS
LIN {X 34.616,Y 50.006,Z -191.883,A 90.000,B 90.000,C 0.000} C_DIS
LIN {X 33.969,Y 50.006,Z -192.445,A 90.000,B 90.000,C 0.000} C_DIS
LIN {X 33.369,Y 50.006,Z -193.059,A 90.000,B 90.000,C 0.000} C_DIS
LIN {X 32.822,Y 50.006,Z -193.718,A 90.000,B 90.000,C 0.000} C_DIS
LIN {X 32.330,Y 50.006,Z -194.420,A 90.000,B 90.000,C 0.000} C_DIS
LIN {X 31.896,Y 50.006,Z -195.160,A 90.000,B 90.000,C 0.000} C_DIS
LIN {X 31.180,Y 50.006,Z -196.083,A 90.000,B 90.000,C 0.000} C_DIS
LIN {X 30.500,Y 50.006,Z -197.033,A 90.000,B 90.000,C 0.000} C_DIS
LIN {X 29.858,Y 50.006,Z -198.008,A 90.000,B 90.000,C 0.000} C_DIS
LIN {X 29.254,Y 50.006,Z -199.009,A 90.000,B 90.000,C 0.000} C_DIS
LIN {X 28.691,Y 50.006,Z -200.032,A 90.000,B 90.000,C 0.000} C_DIS
LIN {X 27.088,Y 50.006,Z -202.466,A 90.000,B 90.000,C 0.000} C_DIS
LIN {X 25.532,Y 50.006,Z -204.930,A 90.000,B 90.000,C 0.000} C_DIS
LIN {X 24.022,Y 50.006,Z -207.422,A 90.000,B 90.000,C 0.000} C_DIS
LIN {X 22.560,Y 50.006,Z -209.943,A 90.000,B 90.000,C 0.000} C_DIS
LIN {X 21.146,Y 50.006,Z -212.491,A 90.000,B 90.000,C 0.000} C_DIS
LIN {X 19.780,Y 50.006,Z -215.066,A 90.000,B 90.000,C 0.000} C_DIS
LIN {X 18.463,Y 50.006,Z -217.665,A 90.000,B 90.000,C 0.000} C_DIS
LIN {X 17.917,Y 50.006,Z -218.730,A 90.000,B 90.000,C 0.000} C_DIS
LIN {X 17.419,Y 50.006,Z -219.819,A 90.000,B 90.000,C 0.000} C_DIS
LIN {X 16.971,Y 50.006,Z -220.929,A 90.000,B 90.000,C 0.000} C_DIS
LIN {X 16.574,Y 50.006,Z -222.058,A 90.000,B 90.000,C 0.000} C_DIS
LIN {X 16.227,Y 50.006,Z -223.203,A 90.000,B 90.000,C 0.000} C_DIS
LIN {X 15.933,Y 50.006,Z -224.364,A 90.000,B 90.000,C 0.000} C_DIS
LIN {X 15.691,Y 50.006,Z -225.536,A 90.000,B 90.000,C 0.000} C_DIS
LIN {X 15.502,Y 50.006,Z -226.718,A 90.000,B 90.000,C 0.000} C_DIS
LIN {X 15.501,Y 50.006,Z -228.182,A 90.000,B 90.000,C 0.000} C_DIS
LIN {X 15.563,Y 50.006,Z -229.644,A 90.000,B 90.000,C 0.000} C_DIS
LIN {X 15.689,Y 50.006,Z -231.102,A 90.000,B 90.000,C 0.000} C_DIS
LIN {X 15.877,Y 50.006,Z -232.553,A 90.000,B 90.000,C 0.000} C_DIS
LIN {X 16.128,Y 50.006,Z -233.995,A 90.000,B 90.000,C 0.000} C_DIS
LIN {X 16.307,Y 50.006,Z -234.740,A 90.000,B 90.000,C 0.000} C_DIS
LIN {X 16.546,Y 50.006,Z -235.469,A 90.000,B 90.000,C 0.000} C_DIS
LIN {X 16.843,Y 50.006,Z -236.176,A 90.000,B 90.000,C 0.000} C_DIS
LIN {X 17.195,Y 50.006,Z -236.857,A 90.000,B 90.000,C 0.000} C_DIS
LIN {X 17.601,Y 50.006,Z -237.507,A 90.000,B 90.000,C 0.000} C_DIS
LIN {X 18.059,Y 50.006,Z -238.123,A 90.000,B 90.000,C 0.000} C_DIS
LIN {X 18.564,Y 50.006,Z -238.700,A 90.000,B 90.000,C 0.000} C_DIS
LIN {X 19.114,Y 50.006,Z -239.234,A 90.000,B 90.000,C 0.000} C_DIS
LIN {X 19.705,Y 50.006,Z -239.722,A 90.000,B 90.000,C 0.000} C_DIS
LIN {X 20.496,Y 50.006,Z -240.207,A 90.000,B 90.000,C 0.000} C_DIS
LIN {X 21.317,Y 50.006,Z -240.637,A 90.000,B 90.000,C 0.000} C_DIS
LIN {X 22.166,Y 50.006,Z -241.010,A 90.000,B 90.000,C 0.000} C_DIS
LIN {X 23.039,Y 50.006,Z -241.324,A 90.000,B 90.000,C 0.000} C_DIS
LIN {X 23.931,Y 50.006,Z -241.579,A 90.000,B 90.000,C 0.000} C_DIS
LIN {X 24.838,Y 50.006,Z -241.772,A 90.000,B 90.000,C 0.000} C_DIS
LIN {X 25.756,Y 50.006,Z -241.903,A 90.000,B 90.000,C 0.000} C_DIS
LIN {X 26.462,Y 50.006,Z -242.145,A 90.000,B 90.000,C 0.000} C_DIS
LIN {X 27.184,Y 50.006,Z -242.335,A 90.000,B 90.000,C 0.000} C_DIS
LIN {X 27.918,Y 50.006,Z -242.472,A 90.000,B 90.000,C 0.000} C_DIS
LIN {X 28.660,Y 50.006,Z -242.556,A 90.000,B 90.000,C 0.000} C_DIS
LIN {X 29.406,Y 50.006,Z -242.585,A 90.000,B 90.000,C 0.000} C_DIS
LIN {X 30.153,Y 50.006,Z -242.561,A 90.000,B 90.000,C 0.000} C_DIS
LIN {X 30.895,Y 50.006,Z -242.483,A 90.000,B 90.000,C 0.000} C_DIS
LIN {X 31.630,Y 50.006,Z -242.351,A 90.000,B 90.000,C 0.000} C_DIS
LIN {X 32.745,Y 50.006,Z -241.989,A 90.000,B 90.000,C 0.000} C_DIS
LIN {X 33.839,Y 50.006,Z -241.571,A 90.000,B 90.000,C 0.000} C_DIS
LIN {X 34.911,Y 50.006,Z -241.097,A 90.000,B 90.000,C 0.000} C_DIS
LIN {X 35.957,Y 50.006,Z -240.569,A 90.000,B 90.000,C 0.000} C_DIS
LIN {X 36.975,Y 50.006,Z -239.989,A 90.000,B 90.000,C 0.000} C_DIS
LIN {X 37.961,Y 50.006,Z -239.357,A 90.000,B 90.000,C 0.000} C_DIS
LIN {X 38.914,Y 50.006,Z -238.675,A 90.000,B 90.000,C 0.000} C_DIS
LIN {X 39.831,Y 50.006,Z -237.945,A 90.000,B 90.000,C 0.000} C_DIS
LIN {X 40.710,Y 50.006,Z -237.170,A 90.000,B 90.000,C 0.000} C_DIS
LIN {X 41.547,Y 50.006,Z -236.350,A 90.000,B 90.000,C 0.000} C_DIS
LIN {X 44.413,Y 50.006,Z -233.448,A 90.000,B 90.000,C 0.000} C_DIS
LIN {X 45.329,Y 50.006,Z -232.188,A 90.000,B 90.000,C 0.000} C_DIS
LIN {X 46.195,Y 50.006,Z -230.893,A 90.000,B 90.000,C 0.000} C_DIS
LIN {X 47.012,Y 50.006,Z -229.567,A 90.000,B 90.000,C 0.000} C_DIS
LIN {X 47.778,Y 50.006,Z -228.210,A 90.000,B 90.000,C 0.000} C_DIS
LIN {X 48.492,Y 50.006,Z -226.826,A 90.000,B 90.000,C 0.000} C_DIS
LIN {X 49.152,Y 50.006,Z -225.415,A 90.000,B 90.000,C 0.000} C_DIS
LIN {X 49.758,Y 50.006,Z -223.980,A 90.000,B 90.000,C 0.000} C_DIS
LIN {X 50.310,Y 50.006,Z -222.523,A 90.000,B 90.000,C 0.000} C_DIS
LIN {X 50.805,Y 50.006,Z -221.046,A 90.000,B 90.000,C 0.000} C_DIS
LIN {X 51.243,Y 50.006,Z -219.551,A 90.000,B 90.000,C 0.000} C_DIS
LIN {X 52.219,Y 50.006,Z -215.738,A 90.000,B 90.000,C 0.000} C_DIS
LIN {X 53.228,Y 50.006,Z -211.933,A 90.000,B 90.000,C 0.000} C_DIS
LIN {X 54.270,Y 50.006,Z -208.137,A 90.000,B 90.000,C 0.000} C_DIS
LIN {X 54.491,Y 50.006,Z -207.425,A 90.000,B 90.000,C 0.000} C_DIS
LIN {X 54.660,Y 50.006,Z -206.700,A 90.000,B 90.000,C 0.000} C_DIS
LIN {X 54.778,Y 50.006,Z -205.964,A 90.000,B 90.000,C 0.000} C_DIS
LIN {X 54.842,Y 50.006,Z -205.221,A 90.000,B 90.000,C 0.000} C_DIS
LIN {X 54.854,Y 50.006,Z -204.476,A 90.000,B 90.000,C 0.000} C_DIS
LIN {X 54.812,Y 50.006,Z -203.732,A 90.000,B 90.000,C 0.000} C_DIS
LIN {X 54.716,Y 50.006,Z -203.252,A 90.000,B 90.000,C 0.000} C_DIS
LIN {X 54.653,Y 50.006,Z -202.767,A 90.000,B 90.000,C 0.000} C_DIS
LIN {X 54.623,Y 50.006,Z -202.278,A 90.000,B 90.000,C 0.000} C_DIS
LIN {X 54.625,Y 50.006,Z -201.789,A 90.000,B 90.000,C 0.000} C_DIS
LIN {X 54.511,Y 50.006,Z -200.547,A 90.000,B 90.000,C 0.000} C_DIS
LIN {X 54.431,Y 50.006,Z -199.302,A 90.000,B 90.000,C 0.000} C_DIS
LIN {X 54.384,Y 50.006,Z -198.055,A 90.000,B 90.000,C 0.000} C_DIS
LIN {X 54.371,Y 50.006,Z -196.808,A 90.000,B 90.000,C 0.000} C_DIS
LIN {X 54.257,Y 50.006,Z -196.004,A 90.000,B 90.000,C 0.000} C_DIS
LIN {X 54.076,Y 50.006,Z -195.213,A 90.000,B 90.000,C 0.000} C_DIS
LIN {X 53.827,Y 50.006,Z -194.440,A 90.000,B 90.000,C 0.000} C_DIS
LIN {X 53.514,Y 50.006,Z -193.691,A 90.000,B 90.000,C 0.000} C_DIS
LIN {X 53.138,Y 50.006,Z -192.971,A 90.000,B 90.000,C 0.000} C_DIS
LIN {X 52.702,Y 50.006,Z -192.286,A 90.000,B 90.000,C 0.000} C_DIS
LIN {X 52.209,Y 50.006,Z -191.641,A 90.000,B 90.000,C 0.000} C_DIS
LIN {X 51.663,Y 50.006,Z -191.040,A 90.000,B 90.000,C 0.000} C_DIS
LIN {X 51.068,Y 50.006,Z -190.488,A 90.000,B 90.000,C 0.000} C_DIS
LIN {X 50.428,Y 50.006,Z -189.988,A 90.000,B 90.000,C 0.000} C_DIS
LIN {X 49.748,Y 50.006,Z -189.545,A 90.000,B 90.000,C 0.000} C_DIS
LIN {X 49.033,Y 50.006,Z -189.161,A 90.000,B 90.000,C 0.000} C_DIS
LIN {X 48.287,Y 50.006,Z -188.839,A 90.000,B 90.000,C 0.000} C_DIS
LIN {X 47.517,Y 50.006,Z -188.583,A 90.000,B 90.000,C 0.000} C_DIS
LIN {X 46.728,Y 50.006,Z -188.392,A 90.000,B 90.000,C 0.000} C_DIS
LIN {X 45.925,Y 50.006,Z -188.270,A 90.000,B 90.000,C 0.000} C_DIS
LIN {X 45.115,Y 50.006,Z -188.217,A 90.000,B 90.000,C 0.000} C_DIS
LIN {X 44.102,Y 50.006,Z -188.315,A 90.000,B 90.000,C 0.000} C_DIS
LIN {X 43.098,Y 50.006,Z -188.477,A 90.000,B 90.000,C 0.000} C_DIS
LIN {X 42.106,Y 50.006,Z -188.703,A 90.000,B 90.000,C 0.000} C_DIS
LIN {X 41.130,Y 50.006,Z -188.993,A 90.000,B 90.000,C 0.000} C_DIS
LIN {X 40.175,Y 50.006,Z -189.344,A 90.000,B 90.000,C 0.000} C_DIS
LIN {X 39.245,Y 50.006,Z -189.756,A 90.000,B 90.000,C 0.000} C_DIS
LIN {X 38.410,Y 50.006,Z -189.949,A 90.000,B 90.000,C 0.000} C_DIS
LIN {X 37.593,Y 50.006,Z -190.210,A 90.000,B 90.000,C 0.000} C_DIS
LIN {X 36.800,Y 50.006,Z -190.536,A 90.000,B 90.000,C 0.000} C_DIS
LIN {X 36.036,Y 50.006,Z -190.925,A 90.000,B 90.000,C 0.000} C_DIS
LIN {X 35.306,Y 50.006,Z -191.375,A 90.000,B 90.000,C 0.000} C_DIS
LIN {X 34.616,Y 50.006,Z -191.883,A 90.000,B 90.000,C 0.000} C_DIS
LIN {X 33.969,Y 50.006,Z -192.445,A 90.000,B 90.000,C 0.000} C_DIS
LIN {X 33.369,Y 50.006,Z -193.059,A 90.000,B 90.000,C 0.000} C_DIS
LIN {X 32.822,Y 50.006,Z -193.718,A 90.000,B 90.000,C 0.000} C_DIS
LIN {X 32.330,Y 50.006,Z -194.420,A 90.000,B 90.000,C 0.000} C_DIS
LIN {X 31.896,Y 50.006,Z -195.160,A 90.000,B 90.000,C 0.000} C_DIS
LIN {X 31.180,Y 50.006,Z -196.083,A 90.000,B 90.000,C 0.000} C_DIS
LIN {X 30.500,Y 50.006,Z -197.033,A 90.000,B 90.000,C 0.000} C_DIS
LIN {X 29.858,Y 50.006,Z -198.008,A 90.000,B 90.000,C 0.000} C_DIS
LIN {X 29.254,Y 50.006,Z -199.009,A 90.000,B 90.000,C 0.000} C_DIS
LIN {X 28.691,Y 50.006,Z -200.032,A 90.000,B 90.000,C 0.000} C_DIS
LIN {X 27.412,Y 50.006,Z -201.967,A 90.000,B 90.000,C 0.000} C_DIS
LIN {X 26.161,Y 50.006,Z -203.920,A 90.000,B 90.000,C 0.000} C_DIS
LIN {X -21.685,Y 50.006,Z -243.561,A 90.000,B 90.000,C 0.000} C_DIS
LIN {X -22.445,Y 50.006,Z -242.471,A 90.000,B 90.000,C 0.000} C_DIS
LIN {X -23.244,Y 50.006,Z -241.409,A 90.000,B 90.000,C 0.000} C_DIS
LIN {X -24.079,Y 50.006,Z -240.375,A 90.000,B 90.000,C 0.000} C_DIS
LIN {X -24.951,Y 50.006,Z -239.372,A 90.000,B 90.000,C 0.000} C_DIS
LIN {X -25.858,Y 50.006,Z -238.400,A 90.000,B 90.000,C 0.000} C_DIS
LIN {X -26.799,Y 50.006,Z -237.462,A 90.000,B 90.000,C 0.000} C_DIS
LIN {X -27.874,Y 50.006,Z -236.699,A 90.000,B 90.000,C 0.000} C_DIS
LIN {X -28.983,Y 50.006,Z -235.986,A 90.000,B 90.000,C 0.000} C_DIS
LIN {X -30.122,Y 50.006,Z -235.324,A 90.000,B 90.000,C 0.000} C_DIS
LIN {X -31.291,Y 50.006,Z -234.714,A 90.000,B 90.000,C 0.000} C_DIS
LIN {X -32.486,Y 50.006,Z -234.158,A 90.000,B 90.000,C 0.000} C_DIS
LIN {X -33.736,Y 50.006,Z -233.770,A 90.000,B 90.000,C 0.000} C_DIS
LIN {X -35.004,Y 50.006,Z -233.445,A 90.000,B 90.000,C 0.000} C_DIS
LIN {X -36.287,Y 50.006,Z -233.183,A 90.000,B 90.000,C 0.000} C_DIS
LIN {X -37.581,Y 50.006,Z -232.984,A 90.000,B 90.000,C 0.000} C_DIS
LIN {X -38.883,Y 50.006,Z -232.850,A 90.000,B 90.000,C 0.000} C_DIS
LIN {X -40.190,Y 50.006,Z -232.780,A 90.000,B 90.000,C 0.000} C_DIS
LIN {X -41.710,Y 50.006,Z -232.795,A 90.000,B 90.000,C 0.000} C_DIS
LIN {X -43.229,Y 50.006,Z -232.868,A 90.000,B 90.000,C 0.000} C_DIS
LIN {X -44.743,Y 50.006,Z -232.996,A 90.000,B 90.000,C 0.000} C_DIS
LIN {X -46.252,Y 50.006,Z -233.182,A 90.000,B 90.000,C 0.000} C_DIS
LIN {X -47.753,Y 50.006,Z -233.423,A 90.000,B 90.000,C 0.000} C_DIS
LIN {X -49.244,Y 50.006,Z -233.720,A 90.000,B 90.000,C 0.000} C_DIS
LIN {X -50.723,Y 50.006,Z -234.073,A 90.000,B 90.000,C 0.000} C_DIS
LIN {X -53.095,Y 50.006,Z -234.786,A 90.000,B 90.000,C 0.000} C_DIS
LIN {X -55.452,Y 50.006,Z -235.549,A 90.000,B 90.000,C 0.000} C_DIS
LIN {X -57.792,Y 50.006,Z -236.360,A 90.000,B 90.000,C 0.000} C_DIS
LIN {X -60.116,Y 50.006,Z -237.218,A 90.000,B 90.000,C 0.000} C_DIS
LIN {X -62.842,Y 50.006,Z -238.380,A 90.000,B 90.000,C 0.000} C_DIS
LIN {X -65.544,Y 50.006,Z -239.595,A 90.000,B 90.000,C 0.000} C_DIS
LIN {X -68.221,Y 50.006,Z -240.864,A 90.000,B 90.000,C 0.000} C_DIS
LIN {X -70.872,Y 50.006,Z -242.187,A 90.000,B 90.000,C 0.000} C_DIS
LIN {X -73.497,Y 50.006,Z -243.561,A 90.000,B 90.000,C 0.000} C_DIS
LIN {X -145.015,Y 50.006,Z -243.561,A 90.000,B 90.000,C 0.000} C_DIS
LIN {X -145.015,Y 50.006,Z 0.000,A 90.000,B 90.000,C 0.000} C_DIS
LIN {X 145.015,Y 50.006,Z 0.000,A 90.000,B 90.000,C 0.000} C_DIS
LIN {X 145.015,Y 50.006,Z -243.561,A 90.000,B 90.000,C 0.000} C_DIS
LIN {X -21.685,Y 50.006,Z -243.561,A 90.000,B 90.000,C 0.000} C_DIS
LIN {X 83.775,Y 50.006,Z -76.746,A 90.000,B 90.000,C 0.000} C_DIS
LIN {X 84.602,Y 50.006,Z -77.205,A 90.000,B 90.000,C 0.000} C_DIS
LIN {X 85.458,Y 50.006,Z -77.608,A 90.000,B 90.000,C 0.000} C_DIS
LIN {X 86.337,Y 50.006,Z -77.956,A 90.000,B 90.000,C 0.000} C_DIS
LIN {X 87.238,Y 50.006,Z -78.245,A 90.000,B 90.000,C 0.000} C_DIS
LIN {X 88.156,Y 50.006,Z -78.475,A 90.000,B 90.000,C 0.000} C_DIS
LIN {X 89.086,Y 50.006,Z -78.645,A 90.000,B 90.000,C 0.000} C_DIS
LIN {X 89.191,Y 50.006,Z -78.671,A 90.000,B 90.000,C 0.000} C_DIS
LIN {X 90.153,Y 50.006,Z -78.809,A 90.000,B 90.000,C 0.000} C_DIS
LIN {X 91.120,Y 50.006,Z -78.897,A 90.000,B 90.000,C 0.000} C_DIS
LIN {X 92.091,Y 50.006,Z -78.933,A 90.000,B 90.000,C 0.000} C_DIS
LIN {X 93.063,Y 50.006,Z -78.918,A 90.000,B 90.000,C 0.000} C_DIS
LIN {X 94.182,Y 50.006,Z -78.787,A 90.000,B 90.000,C 0.000} C_DIS
LIN {X 95.292,Y 50.006,Z -78.590,A 90.000,B 90.000,C 0.000} C_DIS
LIN {X 96.387,Y 50.006,Z -78.326,A 90.000,B 90.000,C 0.000} C_DIS
LIN {X 97.465,Y 50.006,Z -77.998,A 90.000,B 90.000,C 0.000} C_DIS
LIN {X 98.521,Y 50.006,Z -77.606,A 90.000,B 90.000,C 0.000} C_DIS
LIN {X 99.552,Y 50.006,Z -77.152,A 90.000,B 90.000,C 0.000} C_DIS
LIN {X 100.555,Y 50.006,Z -76.636,A 90.000,B 90.000,C 0.000} C_DIS
LIN {X 101.524,Y 50.006,Z -76.062,A 90.000,B 90.000,C 0.000} C_DIS
LIN {X 102.458,Y 50.006,Z -75.431,A 90.000,B 90.000,C 0.000} C_DIS
LIN {X 103.352,Y 50.006,Z -74.745,A 90.000,B 90.000,C 0.000} C_DIS
LIN {X 104.203,Y 50.006,Z -74.008,A 90.000,B 90.000,C 0.000} C_DIS
LIN {X 105.009,Y 50.006,Z -73.220,A 90.000,B 90.000,C 0.000} C_DIS
LIN {X 105.767,Y 50.006,Z -72.386,A 90.000,B 90.000,C 0.000} C_DIS
LIN {X 106.732,Y 50.006,Z -71.227,A 90.000,B 90.000,C 0.000} C_DIS
LIN {X 107.644,Y 50.006,Z -70.025,A 90.000,B 90.000,C 0.000} C_DIS
LIN {X 108.501,Y 50.006,Z -68.783,A 90.000,B 90.000,C 0.000} C_DIS
LIN {X 109.300,Y 50.006,Z -67.503,A 90.000,B 90.000,C 0.000} C_DIS
LIN {X 110.040,Y 50.006,Z -66.189,A 90.000,B 90.000,C 0.000} C_DIS
LIN {X 110.721,Y 50.006,Z -64.843,A 90.000,B 90.000,C 0.000} C_DIS
LIN {X 111.339,Y 50.006,Z -63.467,A 90.000,B 90.000,C 0.000} C_DIS
LIN {X 111.895,Y 50.006,Z -62.064,A 90.000,B 90.000,C 0.000} C_DIS
LIN {X 112.387,Y 50.006,Z -60.638,A 90.000,B 90.000,C 0.000} C_DIS
LIN {X 112.813,Y 50.006,Z -59.191,A 90.000,B 90.000,C 0.000} C_DIS
LIN {X 113.174,Y 50.006,Z -57.726,A 90.000,B 90.000,C 0.000} C_DIS
LIN {X 113.467,Y 50.006,Z -56.246,A 90.000,B 90.000,C 0.000} C_DIS
LIN {X 113.586,Y 50.006,Z -54.778,A 90.000,B 90.000,C 0.000} C_DIS
LIN {X 113.748,Y 50.006,Z -53.314,A 90.000,B 90.000,C 0.000} C_DIS
LIN {X 113.952,Y 50.006,Z -51.855,A 90.000,B 90.000,C 0.000} C_DIS
LIN {X 114.062,Y 50.006,Z -50.984,A 90.000,B 90.000,C 0.000} C_DIS
LIN {X 114.144,Y 50.006,Z -50.109,A 90.000,B 90.000,C 0.000} C_DIS
LIN {X 114.200,Y 50.006,Z -49.233,A 90.000,B 90.000,C 0.000} C_DIS
LIN {X 114.239,Y 50.006,Z -48.325,A 90.000,B 90.000,C 0.000} C_DIS
LIN {X 114.202,Y 50.006,Z -47.417,A 90.000,B 90.000,C 0.000} C_DIS
LIN {X 114.090,Y 50.006,Z -46.516,A 90.000,B 90.000,C 0.000} C_DIS
LIN {X 113.904,Y 50.006,Z -45.627,A 90.000,B 90.000,C 0.000} C_DIS
LIN {X 113.645,Y 50.006,Z -44.756,A 90.000,B 90.000,C 0.000} C_DIS
LIN {X 113.314,Y 50.006,Z -43.910,A 90.000,B 90.000,C 0.000} C_DIS
LIN {X 112.915,Y 50.006,Z -43.094,A 90.000,B 90.000,C 0.000} C_DIS
LIN {X 112.449,Y 50.006,Z -42.314,A 90.000,B 90.000,C 0.000} C_DIS
LIN {X 111.920,Y 50.006,Z -41.575,A 90.000,B 90.000,C 0.000} C_DIS
LIN {X 111.331,Y 50.006,Z -40.883,A 90.000,B 90.000,C 0.000} C_DIS
LIN {X 110.687,Y 50.006,Z -40.242,A 90.000,B 90.000,C 0.000} C_DIS
LIN {X 109.992,Y 50.006,Z -39.656,A 90.000,B 90.000,C 0.000} C_DIS
LIN {X 109.251,Y 50.006,Z -39.131,A 90.000,B 90.000,C 0.000} C_DIS
LIN {X 108.469,Y 50.006,Z -38.668,A 90.000,B 90.000,C 0.000} C_DIS
LIN {X 107.652,Y 50.006,Z -38.272,A 90.000,B 90.000,C 0.000} C_DIS
LIN {X 106.804,Y 50.006,Z -37.945,A 90.000,B 90.000,C 0.000} C_DIS
LIN {X 105.932,Y 50.006,Z -37.690,A 90.000,B 90.000,C 0.000} C_DIS
LIN {X 105.042,Y 50.006,Z -37.508,A 90.000,B 90.000,C 0.000} C_DIS
LIN {X 104.140,Y 50.006,Z -37.400,A 90.000,B 90.000,C 0.000} C_DIS
LIN {X 103.232,Y 50.006,Z -37.367,A 90.000,B 90.000,C 0.000} C_DIS
LIN {X 102.324,Y 50.006,Z -37.410,A 90.000,B 90.000,C 0.000} C_DIS
LIN {X 101.424,Y 50.006,Z -37.528,A 90.000,B 90.000,C 0.000} C_DIS
LIN {X 100.536,Y 50.006,Z -37.720,A 90.000,B 90.000,C 0.000} C_DIS
LIN {X 99.667,Y 50.006,Z -37.987,A 90.000,B 90.000,C 0.000} C_DIS
LIN {X 98.729,Y 50.006,Z -38.379,A 90.000,B 90.000,C 0.000} C_DIS
LIN {X 97.810,Y 50.006,Z -38.813,A 90.000,B 90.000,C 0.000} C_DIS
LIN {X 96.910,Y 50.006,Z -39.287,A 90.000,B 90.000,C 0.000} C_DIS
LIN {X 96.033,Y 50.006,Z -39.801,A 90.000,B 90.000,C 0.000} C_DIS
LIN {X 95.180,Y 50.006,Z -40.353,A 90.000,B 90.000,C 0.000} C_DIS
LIN {X 94.352,Y 50.006,Z -40.943,A 90.000,B 90.000,C 0.000} C_DIS
LIN {X 92.367,Y 50.006,Z -42.738,A 90.000,B 90.000,C 0.000} C_DIS
LIN {X 90.353,Y 50.006,Z -44.500,A 90.000,B 90.000,C 0.000} C_DIS
LIN {X 88.311,Y 50.006,Z -46.229,A 90.000,B 90.000,C 0.000} C_DIS
LIN {X 86.874,Y 50.006,Z -47.376,A 90.000,B 90.000,C 0.000} C_DIS
LIN {X 85.477,Y 50.006,Z -48.571,A 90.000,B 90.000,C 0.000} C_DIS
LIN {X 84.121,Y 50.006,Z -49.813,A 90.000,B 90.000,C 0.000} C_DIS
LIN {X 82.807,Y 50.006,Z -51.100,A 90.000,B 90.000,C 0.000} C_DIS
LIN {X 81.539,Y 50.006,Z -52.431,A 90.000,B 90.000,C 0.000} C_DIS
LIN {X 80.316,Y 50.006,Z -53.804,A 90.000,B 90.000,C 0.000} C_DIS
LIN {X 79.667,Y 50.006,Z -54.552,A 90.000,B 90.000,C 0.000} C_DIS
LIN {X 79.064,Y 50.006,Z -55.337,A 90.000,B 90.000,C 0.000} C_DIS
LIN {X 78.510,Y 50.006,Z -56.157,A 90.000,B 90.000,C 0.000} C_DIS
LIN {X 78.006,Y 50.006,Z -57.010,A 90.000,B 90.000,C 0.000} C_DIS
LIN {X 77.554,Y 50.006,Z -57.891,A 90.000,B 90.000,C 0.000} C_DIS
LIN {X 77.157,Y 50.006,Z -58.798,A 90.000,B 90.000,C 0.000} C_DIS
LIN {X 76.815,Y 50.006,Z -59.727,A 90.000,B 90.000,C 0.000} C_DIS
LIN {X 76.530,Y 50.006,Z -60.675,A 90.000,B 90.000,C 0.000} C_DIS
LIN {X 76.276,Y 50.006,Z -61.654,A 90.000,B 90.000,C 0.000} C_DIS
LIN {X 76.097,Y 50.006,Z -62.650,A 90.000,B 90.000,C 0.000} C_DIS
LIN {X 75.992,Y 50.006,Z -63.656,A 90.000,B 90.000,C 0.000} C_DIS
LIN {X 75.964,Y 50.006,Z -64.667,A 90.000,B 90.000,C 0.000} C_DIS
LIN {X 76.012,Y 50.006,Z -65.678,A 90.000,B 90.000,C 0.000} C_DIS
LIN {X 76.136,Y 50.006,Z -66.682,A 90.000,B 90.000,C 0.000} C_DIS
LIN {X 76.334,Y 50.006,Z -67.673,A 90.000,B 90.000,C 0.000} C_DIS
LIN {X 76.607,Y 50.006,Z -68.648,A 90.000,B 90.000,C 0.000} C_DIS
LIN {X 76.952,Y 50.006,Z -69.598,A 90.000,B 90.000,C 0.000} C_DIS
LIN {X 77.368,Y 50.006,Z -70.521,A 90.000,B 90.000,C 0.000} C_DIS
LIN {X 77.852,Y 50.006,Z -71.409,A 90.000,B 90.000,C 0.000} C_DIS
LIN {X 78.401,Y 50.006,Z -72.258,A 90.000,B 90.000,C 0.000} C_DIS
LIN {X 79.013,Y 50.006,Z -73.064,A 90.000,B 90.000,C 0.000} C_DIS
LIN {X 79.683,Y 50.006,Z -73.822,A 90.000,B 90.000,C 0.000} C_DIS
LIN {X 80.409,Y 50.006,Z -74.527,A 90.000,B 90.000,C 0.000} C_DIS
LIN {X 81.185,Y 50.006,Z -75.175,A 90.000,B 90.000,C 0.000} C_DIS
LIN {X 82.008,Y 50.006,Z -75.763,A 90.000,B 90.000,C 0.000} C_DIS
LIN {X 82.873,Y 50.006,Z -76.288,A 90.000,B 90.000,C 0.000} C_DIS
LIN {X 83.775,Y 50.006,Z -76.746,A 90.000,B 90.000,C 0.000} C_DIS
LIN {X 83.775,Y 62.506,Z -76.746,A 90.000,B 90.000,C 0.000} C_DIS
LIN {X 83.775,Y 75.006,Z -76.746,A 90.000,B 90.000,C 0.000} C_DIS
LIN {X 144.015,Y 75.006,Z -242.561,A 90.000,B 90.000,C 0.000} C_DIS
LIN {X 144.015,Y 67.862,Z -242.561,A 90.000,B 90.000,C 0.000} C_DIS
LIN {X 144.015,Y 55.362,Z -242.561,A 90.000,B 90.000,C 0.000} C_DIS
LIN {X 144.015,Y 42.862,Z -242.561,A 90.000,B 90.000,C 0.000} C_DIS
LIN {X 61.890,Y 42.862,Z -242.561,A 90.000,B 90.000,C 0.000} C_DIS
LIN {X 63.275,Y 42.862,Z -240.060,A 90.000,B 90.000,C 0.000} C_DIS
LIN {X 64.631,Y 42.862,Z -237.544,A 90.000,B 90.000,C 0.000} C_DIS
LIN {X 65.959,Y 42.862,Z -235.012,A 90.000,B 90.000,C 0.000} C_DIS
LIN {X 144.015,Y 42.862,Z -235.012,A 90.000,B 90.000,C 0.000} C_DIS
LIN {X 144.015,Y 42.862,Z -227.464,A 90.000,B 90.000,C 0.000} C_DIS
LIN {X 69.705,Y 42.862,Z -227.464,A 90.000,B 90.000,C 0.000} C_DIS
LIN {X 70.879,Y 42.862,Z -224.960,A 90.000,B 90.000,C 0.000} C_DIS
LIN {X 72.025,Y 42.862,Z -222.444,A 90.000,B 90.000,C 0.000} C_DIS
LIN {X 73.143,Y 42.862,Z -219.915,A 90.000,B 90.000,C 0.000} C_DIS
LIN {X 144.015,Y 42.862,Z -219.915,A 90.000,B 90.000,C 0.000} C_DIS
LIN {X 144.015,Y 42.862,Z -212.366,A 90.000,B 90.000,C 0.000} C_DIS
LIN {X 76.287,Y 42.862,Z -212.366,A 90.000,B 90.000,C 0.000} C_DIS
LIN {X 77.254,Y 42.862,Z -209.896,A 90.000,B 90.000,C 0.000} C_DIS
LIN {X 78.194,Y 42.862,Z -207.417,A 90.000,B 90.000,C 0.000} C_DIS
LIN {X 79.108,Y 42.862,Z -204.927,A 90.000,B 90.000,C 0.000} C_DIS
LIN {X 79.153,Y 42.862,Z -204.817,A 90.000,B 90.000,C 0.000} C_DIS
LIN {X 144.015,Y 42.862,Z -204.817,A 90.000,B 90.000,C 0.000} C_DIS
LIN {X 144.015,Y 42.862,Z -197.269,A 90.000,B 90.000,C 0.000} C_DIS
LIN {X 81.859,Y 42.862,Z -197.269,A 90.000,B 90.000,C 0.000} C_DIS
LIN {X 82.492,Y 42.862,Z -195.147,A 90.000,B 90.000,C 0.000} C_DIS
LIN {X 83.076,Y 42.862,Z -193.010,A 90.000,B 90.000,C 0.000} C_DIS
LIN {X 83.609,Y 42.862,Z -190.860,A 90.000,B 90.000,C 0.000} C_DIS
LIN {X 83.850,Y 42.862,Z -189.720,A 90.000,B 90.000,C 0.000} C_DIS
LIN {X 144.015,Y 42.862,Z -189.720,A 90.000,B 90.000,C 0.000} C_DIS
LIN {X 144.015,Y 42.862,Z -182.171,A 90.000,B 90.000,C 0.000} C_DIS
LIN {X 85.701,Y 42.862,Z -182.171,A 90.000,B 90.000,C 0.000} C_DIS
LIN {X 86.269,Y 42.862,Z -180.161,A 90.000,B 90.000,C 0.000} C_DIS
LIN {X 86.867,Y 42.862,Z -178.160,A 90.000,B 90.000,C 0.000} C_DIS
LIN {X 87.495,Y 42.862,Z -176.168,A 90.000,B 90.000,C 0.000} C_DIS
LIN {X 87.766,Y 42.862,Z -175.396,A 90.000,B 90.000,C 0.000} C_DIS
LIN {X 88.032,Y 42.862,Z -174.622,A 90.000,B 90.000,C 0.000} C_DIS
LIN {X 144.015,Y 42.862,Z -174.622,A 90.000,B 90.000,C 0.000} C_DIS
LIN {X 144.015,Y 42.862,Z -167.073,A 90.000,B 90.000,C 0.000} C_DIS
LIN {X 90.296,Y 42.862,Z -167.073,A 90.000,B 90.000,C 0.000} C_DIS
LIN {X 90.769,Y 42.862,Z -165.197,A 90.000,B 90.000,C 0.000} C_DIS
LIN {X 91.210,Y 42.862,Z -163.314,A 90.000,B 90.000,C 0.000} C_DIS
LIN {X 91.617,Y 42.862,Z -161.423,A 90.000,B 90.000,C 0.000} C_DIS
LIN {X 91.992,Y 42.862,Z -159.525,A 90.000,B 90.000,C 0.000} C_DIS
LIN {X 144.015,Y 42.862,Z -159.525,A 90.000,B 90.000,C 0.000} C_DIS
LIN {X 144.015,Y 42.862,Z -151.976,A 90.000,B 90.000,C 0.000} C_DIS
LIN {X 93.146,Y 42.862,Z -151.976,A 90.000,B 90.000,C 0.000} C_DIS
LIN {X 93.405,Y 42.862,Z -149.544,A 90.000,B 90.000,C 0.000} C_DIS
LIN {X 93.611,Y 42.862,Z -147.107,A 90.000,B 90.000,C 0.000} C_DIS
LIN {X 93.763,Y 42.862,Z -144.666,A 90.000,B 90.000,C 0.000} C_DIS
LIN {X 93.769,Y 42.862,Z -144.427,A 90.000,B 90.000,C 0.000} C_DIS
LIN {X 144.015,Y 42.862,Z -144.427,A 90.000,B 90.000,C 0.000} C_DIS
LIN {X 144.015,Y 42.862,Z -136.878,A 90.000,B 90.000,C 0.000} C_DIS
LIN {X 94.065,Y 42.862,Z -136.878,A 90.000,B 90.000,C 0.000} C_DIS
LIN {X 94.249,Y 42.862,Z -133.733,A 90.000,B 90.000,C 0.000} C_DIS
LIN {X 94.470,Y 42.862,Z -130.590,A 90.000,B 90.000,C 0.000} C_DIS
LIN {X 94.532,Y 42.862,Z -129.960,A 90.000,B 90.000,C 0.000} C_DIS
LIN {X 94.580,Y 42.862,Z -129.329,A 90.000,B 90.000,C 0.000} C_DIS
LIN {X 144.015,Y 42.862,Z -129.329,A 90.000,B 90.000,C 0.000} C_DIS
LIN {X 144.015,Y 42.862,Z -121.781,A 90.000,B 90.000,C 0.000} C_DIS
LIN {X 94.029,Y 42.862,Z -121.781,A 90.000,B 90.000,C 0.000} C_DIS
LIN {X 94.006,Y 42.862,Z -121.417,A 90.000,B 90.000,C 0.000} C_DIS
LIN {X 93.800,Y 42.862,Z -120.647,A 90.000,B 90.000,C 0.000} C_DIS
LIN {X 93.644,Y 42.862,Z -119.866,A 90.000,B 90.000,C 0.000} C_DIS
LIN {X 93.538,Y 42.862,Z -119.077,A 90.000,B 90.000,C 0.000} C_DIS
LIN {X 93.898,Y 42.862,Z -118.082,A 90.000,B 90.000,C 0.000} C_DIS
LIN {X 94.224,Y 42.862,Z -117.077,A 90.000,B 90.000,C 0.000} C_DIS
LIN {X 94.517,Y 42.862,Z -116.060,A 90.000,B 90.000,C 0.000} C_DIS
LIN {X 94.776,Y 42.862,Z -115.035,A 90.000,B 90.000,C 0.000} C_DIS
LIN {X 94.792,Y 42.862,Z -114.947,A 90.000,B 90.000,C 0.000} C_DIS
LIN {X 94.973,Y 42.862,Z -114.232,A 90.000,B 90.000,C 0.000} C_DIS
LIN {X 144.015,Y 42.862,Z -114.232,A 90.000,B 90.000,C 0.000} C_DIS
LIN {X 144.015,Y 42.862,Z -106.683,A 90.000,B 90.000,C 0.000} C_DIS
LIN {X 95.979,Y 42.862,Z -106.683,A 90.000,B 90.000,C 0.000} C_DIS
LIN {X 95.928,Y 42.862,Z -105.980,A 90.000,B 90.000,C 0.000} C_DIS
LIN {X 95.852,Y 42.862,Z -105.280,A 90.000,B 90.000,C 0.000} C_DIS
LIN {X 96.426,Y 42.862,Z -104.574,A 90.000,B 90.000,C 0.000} C_DIS
LIN {X 96.957,Y 42.862,Z -103.834,A 90.000,B 90.000,C 0.000} C_DIS
LIN {X 97.443,Y 42.862,Z -103.065,A 90.000,B 90.000,C 0.000} C_DIS
LIN {X 97.883,Y 42.862,Z -102.268,A 90.000,B 90.000,C 0.000} C_DIS
LIN {X 98.274,Y 42.862,Z -101.446,A 90.000,B 90.000,C 0.000} C_DIS
LIN {X 98.615,Y 42.862,Z -100.602,A 90.000,B 90.000,C 0.000} C_DIS
LIN {X 98.905,Y 42.862,Z -99.739,A 90.000,B 90.000,C 0.000} C_DIS
LIN {X 99.063,Y 42.862,Z -99.134,A 90.000,B 90.000,C 0.000} C_DIS
LIN {X 144.015,Y 42.862,Z -99.134,A 90.000,B 90.000,C 0.000} C_DIS
LIN {X 144.015,Y 42.862,Z -91.586,A 90.000,B 90.000,C 0.000} C_DIS
LIN {X 102.044,Y 42.862,Z -91.586,A 90.000,B 90.000,C 0.000} C_DIS
LIN {X 103.211,Y 42.862,Z -90.423,A 90.000,B 90.000,C 0.000} C_DIS
LIN {X 104.337,Y 42.862,Z -89.220,A 90.000,B 90.000,C 0.000} C_DIS
LIN {X 105.420,Y 42.862,Z -87.978,A 90.000,B 90.000,C 0.000} C_DIS
LIN {X 106.459,Y 42.862,Z -86.699,A 90.000,B 90.000,C 0.000} C_DIS
LIN {X 107.453,Y 42.862,Z -85.385,A 90.000,B 90.000,C 0.000} C_DIS
LIN {X 108.401,Y 42.862,Z -84.037,A 90.000,B 90.000,C 0.000} C_DIS
LIN {X 144.015,Y 42.862,Z -84.037,A 90.000,B 90.000,C 0.000} C_DIS
LIN {X 144.015,Y 42.862,Z -76.488,A 90.000,B 90.000,C 0.000} C_DIS
LIN {X 112.521,Y 42.862,Z -76.488,A 90.000,B 90.000,C 0.000} C_DIS
LIN {X 113.375,Y 42.862,Z -74.626,A 90.000,B 90.000,C 0.000} C_DIS
LIN {X 114.191,Y 42.862,Z -72.747,A 90.000,B 90.000,C 0.000} C_DIS
LIN {X 114.966,Y 42.862,Z -70.851,A 90.000,B 90.000,C 0.000} C_DIS
LIN {X 115.702,Y 42.862,Z -68.939,A 90.000,B 90.000,C 0.000} C_DIS
LIN {X 144.015,Y 42.862,Z -68.939,A 90.000,B 90.000,C 0.000} C_DIS
LIN {X 144.015,Y 42.862,Z -61.390,A 90.000,B 90.000,C 0.000} C_DIS
LIN {X 118.239,Y 42.862,Z -61.390,A 90.000,B 90.000,C 0.000} C_DIS
LIN {X 118.728,Y 42.862,Z -60.079,A 90.000,B 90.000,C 0.000} C_DIS
LIN {X 119.247,Y 42.862,Z -58.780,A 90.000,B 90.000,C 0.000} C_DIS
LIN {X 119.795,Y 42.862,Z -57.492,A 90.000,B 90.000,C 0.000} C_DIS
LIN {X 120.373,Y 42.862,Z -56.218,A 90.000,B 90.000,C 0.000} C_DIS
LIN {X 121.029,Y 42.862,Z -55.040,A 90.000,B 90.000,C 0.000} C_DIS
LIN {X 121.647,Y 42.862,Z -53.841,A 90.000,B 90.000,C 0.000} C_DIS
LIN {X 144.015,Y 42.862,Z -53.841,A 90.000,B 90.000,C 0.000} C_DIS
LIN {X 144.015,Y 42.862,Z -46.293,A 90.000,B 90.000,C 0.000} C_DIS
LIN {X 124.613,Y 42.862,Z -46.293,A 90.000,B 90.000,C 0.000} C_DIS
LIN {X 124.835,Y 42.862,Z -45.383,A 90.000,B 90.000,C 0.000} C_DIS
LIN {X 125.001,Y 42.862,Z -44.462,A 90.000,B 90.000,C 0.000} C_DIS
LIN {X 125.109,Y 42.862,Z -43.532,A 90.000,B 90.000,C 0.000} C_DIS
LIN {X 125.158,Y 42.862,Z -42.597,A 90.000,B 90.000,C 0.000} C_DIS
